C02671=1902.025400,220.027500,-703.720300,90.647653,-0.183346,-0.000000
C02672=1936.034400,220.049100,-703.720300,90.647653,-0.183346,-0.000000
C02673=1947.501800,220.061300,-703.720300,90.647653,-0.183346,-0.000000
C02674=1883.123400,220.069100,-703.720300,90.647653,-0.183346,-0.000000
C02675=2183.365000,220.088300,-703.720300,90.647653,-0.183346,-0.000000
C02676=1917.413700,220.121800,-703.720300,90.647653,-0.183346,-0.000000
C02677=1873.196800,220.137600,-703.720300,90.647653,-0.183346,-0.000000
C02678=2183.234000,220.175800,-703.720300,90.647653,-0.183346,-0.000000
C02679=1859.481200,220.212300,-703.720300,90.647653,-0.183346,-0.000000
C02680=1876.167800,220.252900,-703.720300,90.647653,-0.183346,-0.000000
C02681=2184.784300,220.282900,-703.720300,90.647653,-0.183346,-0.000000
C02682=1857.137100,220.330000,-703.720300,90.647653,-0.183346,-0.000000
C02683=1851.834100,220.481200,-703.720300,90.647653,-0.183346,-0.000000
C02684=1843.863200,220.525500,-703.720300,90.647653,-0.183346,-0.000000
C02685=1838.599500,220.632600,-703.720300,90.647653,-0.183346,-0.000000
C02686=1828.269700,220.740000,-703.720300,90.647653,-0.183346,-0.000000
C02687=1824.941700,220.777500,-703.720300,90.647653,-0.183346,-0.000000
C02688=1794.350900,220.933900,-703.720300,90.647653,-0.183346,-0.000000
C02689=1816.456800,221.034500,-703.720300,90.647653,-0.183346,-0.000000
C02690=1818.517400,221.113300,-703.720300,90.647653,-0.183346,-0.000000
C02691=1794.707900,221.180900,-703.720300,90.647653,-0.183346,-0.000000
C02692=1804.703800,221.313700,-703.720300,90.647653,-0.183346,-0.000000
C02693=1808.802700,221.407900,-703.720300,90.647653,-0.183346,-0.000000
C02694=1797.626000,221.486500,-703.720300,90.647653,-0.183346,-0.000000
C02695=1799.014100,221.558000,-703.720300,90.647653,-0.183346,-0.000000
C02696=1799.493300,221.627400,-753.720300,90.647653,-0.183346,-0.000000
C02697=1803.199100,221.533000,-753.720300,90.647653,-0.183346,-0.000000
C02698=1804.482800,221.440400,-753.720300,90.647653,-0.183346,-0.000000
C02699=1806.656400,221.406800,-753.720300,90.647653,-0.183346,-0.000000
C02700=1812.999200,221.332300,-753.720300,90.647653,-0.183346,-0.000000
C02701=1810.456500,221.261700,-753.720300,90.647653,-0.183346,-0.000000
C02702=1819.601700,221.167700,-753.720300,90.647653,-0.183346,-0.000000
C02703=1828.737100,221.094100,-753.720300,90.647653,-0.183346,-0.000000
C02704=1826.975900,220.979200,-753.720300,90.647653,-0.183346,-0.000000
C02705=1827.057400,220.918400,-753.720300,90.647653,-0.183346,-0.000000
C02706=1840.828400,220.793700,-753.720300,90.647653,-0.183346,-0.000000
C02707=1843.616100,220.652500,-753.720300,90.647653,-0.183346,-0.000000
C02708=1848.358800,220.494700,-753.720300,90.647653,-0.183346,-0.000000
C02709=1855.244300,220.394700,-753.720300,90.647653,-0.183346,-0.000000
C02710=1859.292000,220.310300,-753.720300,90.647653,-0.183346,-0.000000
C02711=1861.936400,220.207200,-753.720300,90.647653,-0.183346,-0.000000
C02712=1863.356300,220.145800,-753.720300,90.647653,-0.183346,-0.000000
C02713=1880.995500,220.085300,-753.720300,90.647653,-0.183346,-0.000000
C02714=1886.645600,220.008400,-753.720300,90.647653,-0.183346,-0.000000
C02715=1888.756600,219.930200,-753.720300,90.647653,-0.183346,-0.000000
C02716=1888.087000,219.894400,-753.720300,90.647653,-0.183346,-0.000000
C02717=1901.700500,219.846400,-753.720300,90.647653,-0.183346,-0.000000
C02718=1899.152700,219.782200,-753.720300,90.647653,-0.183346,-0.000000
C02719=1896.702700,219.751800,-753.720300,90.647653,-0.183346,-0.000000
C02720=2159.599800,219.718700,-753.720300,90.647653,-0.183346,-0.000000
C02721=1898.573400,219.689000,-753.720300,90.647653,-0.183346,-0.000000
C02722=2190.999200,219.661600,-753.720300,90.647653,-0.183346,-0.000000
C02723=1908.414200,219.628500,-753.720300,90.647653,-0.183346,-0.000000
C02724=2178.349900,219.615200,-753.720300,90.647653,-0.183346,-0.000000
C02725=1918.020800,219.596800,-753.720300,90.647653,-0.183346,-0.000000
C02726=2162.631500,219.573400,-753.720300,90.647653,-0.183346,-0.000000
C02727=2163.426800,219.563600,-753.720300,90.647653,-0.183346,-0.000000
C02728=1918.500400,219.534600,-753.720300,90.647653,-0.183346,-0.000000
C02729=2179.089400,219.517700,-753.720300,90.647653,-0.183346,-0.000000
C02730=2153.107500,219.504900,-753.720300,90.647653,-0.183346,-0.000000
C02731=1927.323900,219.499800,-753.720300,90.647653,-0.183346,-0.000000
C02732=1962.897900,219.487000,-753.720300,90.647653,-0.183346,-0.000000
C02733=2152.945000,219.474800,-753.720300,90.647653,-0.183346,-0.000000
C02734=1923.549800,219.465000,-753.720300,90.647653,-0.183346,-0.000000
C02735=2167.654000,219.443400,-753.720300,90.647653,-0.183346,-0.000000
C02736=2127.277400,219.427200,-753.720300,90.647653,-0.183346,-0.000000
C02737=2157.455000,219.411600,-753.720300,90.647653,-0.183346,-0.000000
C02738=2181.610100,219.398800,-753.720300,90.647653,-0.183346,-0.000000
C02739=1942.548000,219.387600,-753.720300,90.647653,-0.183346,-0.000000
C02740=1942.914300,219.375500,-753.720300,90.647653,-0.183346,-0.000000
C02741=2146.459000,219.360600,-753.720300,90.647653,-0.183346,-0.000000
C02742=1943.803100,219.342400,-753.720300,90.647653,-0.183346,-0.000000
C02743=2144.906500,219.324500,-753.720300,90.647653,-0.183346,-0.000000
C02744=1955.055200,219.314300,-753.720300,90.647653,-0.183346,-0.000000
C02745=2126.347200,219.294700,-753.720300,90.647653,-0.183346,-0.000000
C02746=1945.956100,219.289000,-753.720300,90.647653,-0.183346,-0.000000
C02747=1962.818800,219.279900,-753.720300,90.647653,-0.183346,-0.000000
C02748=1984.835000,219.262300,-753.720300,90.647653,-0.183346,-0.000000
C02749=1961.384800,219.248800,-753.720300,90.647653,-0.183346,-0.000000
C02750=2132.790400,219.237600,-753.720300,90.647653,-0.183346,-0.000000
C02751=2000.726200,219.227200,-753.720300,90.647653,-0.183346,-0.000000
C02752=1953.023500,219.217700,-753.720300,90.647653,-0.183346,-0.000000
C02753=2110.038700,219.210900,-753.720300,90.647653,-0.183346,-0.000000
C02754=2009.596400,219.203500,-753.720300,90.647653,-0.183346,-0.000000
C02755=2132.660700,219.194400,-753.720300,90.647653,-0.183346,-0.000000
C02756=2014.251400,219.182900,-753.720300,90.647653,-0.183346,-0.000000
C02757=2125.162500,219.168400,-753.720300,90.647653,-0.183346,-0.000000
C02758=2104.208600,219.149400,-753.720300,90.647653,-0.183346,-0.000000
C02759=2129.301800,219.144000,-753.720300,90.647653,-0.183346,-0.000000
C02760=2071.342900,219.139600,-753.720300,90.647653,-0.183346,-0.000000
C02761=2057.003000,219.115300,-753.720300,90.647653,-0.183346,-0.000000
C02762=2060.754400,219.103200,-753.720300,90.647653,-0.183346,-0.000000
C02763=1975.391800,219.089300,-753.720300,90.647653,-0.183346,-0.000000
C02764=2041.350200,219.082200,-753.720300,90.647653,-0.183346,-0.000000
C02765=2058.370700,219.077800,-753.720300,90.647653,-0.183346,-0.000000
C02766=2014.830600,219.072400,-753.720300,90.647653,-0.183346,-0.000000
C02767=1968.445400,219.059600,-753.720300,90.647653,-0.183346,-0.000000
C02768=2054.250900,219.044000,-753.720300,90.647653,-0.183346,-0.000000
C02769=2104.495100,219.038300,-753.720300,90.647653,-0.183346,-0.000000
C02770=2082.338100,219.029200,-753.720300,90.647653,-0.183346,-0.000000
C02771=2027.175600,219.021400,-753.720300,90.647653,-0.183346,-0.000000
C02772=1997.599100,219.010600,-753.720300,90.647653,-0.183346,-0.000000
C02773=2074.350800,218.995400,-753.720300,90.647653,-0.183346,-0.000000
C02774=2088.675300,218.990300,-753.720300,90.647653,-0.183346,-0.000000
C02775=2052.849400,218.981200,-753.720300,90.647653,-0.183346,-0.000000
C02776=2096.650800,218.977100,-753.720300,90.647653,-0.183346,-0.000000
C02777=2021.793300,218.962300,-753.720300,90.647653,-0.183346,-0.000000
C02778=2024.376200,218.935600,-753.720300,90.647653,-0.183346,-0.000000
C02779=2084.858800,218.917700,-753.720300,90.647653,-0.183346,-0.000000
C02780=2037.732300,218.909600,-753.720300,90.647653,-0.183346,-0.000000
C02781=2066.030000,218.889600,-753.720300,90.647653,-0.183346,-0.000000
C02782=2093.060000,218.868000,-753.720300,90.647653,-0.183346,-0.000000
C02783=2057.961700,218.804300,-753.720300,90.647653,-0.183346,-0.000000
C02784=2072.588600,218.737900,-803.720300,90.647653,-0.183346,-0.000000
C02785=2061.790300,218.784200,-803.720300,90.647653,-0.183346,-0.000000
C02786=2060.744300,218.794000,-803.720300,90.647653,-0.183346,-0.000000
C02787=1998.766800,218.818700,-803.720300,90.647653,-0.183346,-0.000000
C02788=2060.686400,218.861300,-803.720300,90.647653,-0.183346,-0.000000
C02789=2096.522100,218.870400,-803.720300,90.647653,-0.183346,-0.000000
C02790=2032.427400,218.885600,-803.720300,90.647653,-0.183346,-0.000000
C02791=2103.743000,218.891700,-803.720300,90.647653,-0.183346,-0.000000
C02792=2019.306500,218.901100,-803.720300,90.647653,-0.183346,-0.000000
C02793=2031.745000,218.913300,-803.720300,90.647653,-0.183346,-0.000000
C02794=2088.498600,218.920400,-803.720300,90.647653,-0.183346,-0.000000
C02795=2037.798100,218.927100,-803.720300,90.647653,-0.183346,-0.000000
C02796=2014.134600,218.935900,-803.720300,90.647653,-0.183346,-0.000000
C02797=2099.616700,218.942000,-803.720300,90.647653,-0.183346,-0.000000
C02798=2045.679500,218.947800,-803.720300,90.647653,-0.183346,-0.000000
C02799=2076.855800,218.951800,-803.720300,90.647653,-0.183346,-0.000000
C02800=2071.493100,218.956200,-803.720300,90.647653,-0.183346,-0.000000
C02801=1988.395700,218.967300,-803.720300,90.647653,-0.183346,-0.000000
C02802=2111.290700,218.977500,-803.720300,90.647653,-0.183346,-0.000000
C02803=2118.179700,218.990000,-803.720300,90.647653,-0.183346,-0.000000
C02804=2105.312500,218.993700,-803.720300,90.647653,-0.183346,-0.000000
C02805=2049.201500,218.998800,-803.720300,90.647653,-0.183346,-0.000000
C02806=2122.327100,219.005500,-803.720300,90.647653,-0.183346,-0.000000
C02807=1998.043700,219.019700,-803.720300,90.647653,-0.183346,-0.000000
C02808=2158.716300,219.030900,-803.720300,90.647653,-0.183346,-0.000000
C02809=2101.906500,219.037600,-803.720300,90.647653,-0.183346,-0.000000
C02810=2041.862200,219.043400,-803.720300,90.647653,-0.183346,-0.000000
C02811=2113.073500,219.050500,-803.720300,90.647653,-0.183346,-0.000000
C02812=2130.536300,219.062600,-803.720300,90.647653,-0.183346,-0.000000
C02813=1989.990900,219.069400,-803.720300,90.647653,-0.183346,-0.000000
C02814=2153.711100,219.082200,-803.720300,90.647653,-0.183346,-0.000000
C02815=2103.281100,219.093000,-803.720300,90.647653,-0.183346,-0.000000
C02816=1978.401700,219.105400,-803.720300,90.647653,-0.183346,-0.000000
C02817=2108.215500,219.112300,-803.720300,90.647653,-0.183346,-0.000000
C02818=2116.807500,219.121100,-803.720300,90.647653,-0.183346,-0.000000
C02819=2167.389500,219.129500,-803.720300,90.647653,-0.183346,-0.000000
C02820=1968.224900,219.147100,-803.720300,90.647653,-0.183346,-0.000000
C02821=1980.356400,219.152100,-803.720300,90.647653,-0.183346,-0.000000
C02822=2012.286700,219.161300,-803.720300,90.647653,-0.183346,-0.000000
C02823=1979.045200,219.176100,-803.720300,90.647653,-0.183346,-0.000000
C02824=2132.626900,219.183900,-803.720300,90.647653,-0.183346,-0.000000
C02825=2138.833300,219.206700,-803.720300,90.647653,-0.183346,-0.000000
C02826=2189.419500,219.215000,-803.720300,90.647653,-0.183346,-0.000000
C02827=2163.932900,219.221100,-803.720300,90.647653,-0.183346,-0.000000
C02828=1973.290700,219.229500,-803.720300,90.647653,-0.183346,-0.000000
C02829=1962.589400,219.234900,-803.720300,90.647653,-0.183346,-0.000000
C02830=2140.348900,219.251500,-803.720300,90.647653,-0.183346,-0.000000
C02831=1966.086800,219.259900,-803.720300,90.647653,-0.183346,-0.000000
C02832=2146.072100,219.278200,-803.720300,90.647653,-0.183346,-0.000000
C02833=1944.019200,219.307900,-803.720300,90.647653,-0.183346,-0.000000
C02834=2164.122900,219.335600,-803.720300,90.647653,-0.183346,-0.000000
C02835=2179.267500,219.347800,-803.720300,90.647653,-0.183346,-0.000000
C02836=1958.782200,219.356200,-803.720300,90.647653,-0.183346,-0.000000
C02837=1950.731800,219.377800,-803.720300,90.647653,-0.183346,-0.000000
C02838=1939.923400,219.405900,-803.720300,90.647653,-0.183346,-0.000000
C02839=1952.384300,219.433200,-803.720300,90.647653,-0.183346,-0.000000
C02840=1939.916500,219.453500,-803.720300,90.647653,-0.183346,-0.000000
C02841=1924.529600,219.509300,-803.720300,90.647653,-0.183346,-0.000000
C02842=1931.308400,219.530200,-803.720300,90.647653,-0.183346,-0.000000
C02843=1915.280200,219.568700,-803.720300,90.647653,-0.183346,-0.000000
C02844=1925.417000,219.624800,-803.720300,90.647653,-0.183346,-0.000000
C02845=1938.538700,219.697400,-803.720300,90.647653,-0.183346,-0.000000
C02846=1916.231700,219.759600,-803.720300,90.647653,-0.183346,-0.000000
C02847=1905.662800,219.803200,-803.720300,90.647653,-0.183346,-0.000000
C02848=1907.860700,219.882600,-803.720300,90.647653,-0.183346,-0.000000
C02849=1891.452900,219.963300,-803.720300,90.647653,-0.183346,-0.000000
C02850=1897.806200,220.044700,-803.720300,90.647653,-0.183346,-0.000000
C02851=1877.774400,220.141500,-803.720300,90.647653,-0.183346,-0.000000
C02852=1889.906800,220.208900,-803.720300,90.647653,-0.183346,-0.000000
C02853=1873.599400,220.241000,-803.720300,90.647653,-0.183346,-0.000000
C02854=1871.595600,220.341000,-803.720300,90.647653,-0.183346,-0.000000
C02855=1877.964600,220.428500,-803.720300,90.647653,-0.183346,-0.000000
C02856=1863.088700,220.547800,-803.720300,90.647653,-0.183346,-0.000000
C02857=1857.730100,220.604900,-803.720300,90.647653,-0.183346,-0.000000
C02858=1845.662400,220.779600,-803.720300,90.647653,-0.183346,-0.000000
C02859=1845.976100,220.851500,-803.720300,90.647653,-0.183346,-0.000000
C02860=1839.138000,220.982300,-803.720300,90.647653,-0.183346,-0.000000
C02861=1829.338300,221.025500,-803.720300,90.647653,-0.183346,-0.000000
C02862=1794.450600,221.067700,-803.720300,90.647653,-0.183346,-0.000000
C02863=1837.453500,221.120100,-803.720300,90.647653,-0.183346,-0.000000
C02864=1823.782100,221.184000,-803.720300,90.647653,-0.183346,-0.000000
C02865=1816.928300,221.265000,-803.720300,90.647653,-0.183346,-0.000000
C02866=1816.898000,221.328600,-803.720300,90.647653,-0.183346,-0.000000
C02867=1807.872100,221.425900,-803.720300,90.647653,-0.183346,-0.000000
C02868=1812.030900,221.466400,-803.720300,90.647653,-0.183346,-0.000000
C02869=1797.540300,221.537700,-803.720300,90.647653,-0.183346,-0.000000
C02870=1797.919500,221.574000,-803.720300,90.647653,-0.183346,-0.000000
C02871=1798.307500,221.652200,-803.720300,90.647653,-0.183346,-0.000000
C02872=1798.204800,221.824500,-853.720300,90.647653,-0.183346,-0.000000
C02873=1801.321900,221.694400,-853.720300,90.647653,-0.183346,-0.000000
C02874=1803.359500,221.606900,-853.720300,90.647653,-0.183346,-0.000000
C02875=1796.778200,221.518400,-853.720300,90.647653,-0.183346,-0.000000
C02876=1810.824300,221.446100,-853.720300,90.647653,-0.183346,-0.000000
C02877=1812.569900,221.372100,-853.720300,90.647653,-0.183346,-0.000000
C02878=1813.958700,221.320100,-853.720300,90.647653,-0.183346,-0.000000
C02879=1816.060500,221.201900,-853.720300,90.647653,-0.183346,-0.000000
C02880=1822.471300,221.136300,-853.720300,90.647653,-0.183346,-0.000000
C02881=1816.917900,221.114700,-853.720300,90.647653,-0.183346,-0.000000
C02882=1843.384000,220.988000,-853.720300,90.647653,-0.183346,-0.000000
C02883=1841.543700,220.882300,-853.720300,90.647653,-0.183346,-0.000000
C02884=1842.988700,220.787700,-853.720300,90.647653,-0.183346,-0.000000
C02885=1849.877000,220.765400,-853.720300,90.647653,-0.183346,-0.000000
C02886=1858.351200,220.668100,-853.720300,90.647653,-0.183346,-0.000000
C02887=1864.384500,220.598800,-853.720300,90.647653,-0.183346,-0.000000
C02888=1864.226300,220.572800,-853.720300,90.647653,-0.183346,-0.000000
C02889=1884.340500,220.452200,-853.720300,90.647653,-0.183346,-0.000000
C02890=1866.225600,220.418700,-853.720300,90.647653,-0.183346,-0.000000
C02891=1874.781700,220.325800,-853.720300,90.647653,-0.183346,-0.000000
C02892=1888.846900,220.302500,-853.720300,90.647653,-0.183346,-0.000000
C02893=1890.867400,220.245800,-853.720300,90.647653,-0.183346,-0.000000
C02894=1896.806300,220.168700,-853.720300,90.647653,-0.183346,-0.000000
C02895=1904.238600,220.121800,-853.720300,90.647653,-0.183346,-0.000000
C02896=1933.711600,220.093100,-853.720300,90.647653,-0.183346,-0.000000
C02897=1904.412600,220.009600,-853.720300,90.647653,-0.183346,-0.000000
C02898=1912.942200,219.983900,-853.720300,90.647653,-0.183346,-0.000000
C02899=1923.653300,219.915300,-853.720300,90.647653,-0.183346,-0.000000
C02900=1952.154200,219.830900,-853.720300,90.647653,-0.183346,-0.000000
C02901=1953.177900,219.787300,-853.720300,90.647653,-0.183346,-0.000000
C02902=1946.822900,219.765300,-853.720300,90.647653,-0.183346,-0.000000
C02903=1929.570200,219.735600,-853.720300,90.647653,-0.183346,-0.000000
C02904=1937.309500,219.673800,-853.720300,90.647653,-0.183346,-0.000000
C02905=1937.928700,219.640000,-853.720300,90.647653,-0.183346,-0.000000
C02906=2046.786800,219.592700,-853.720300,90.647653,-0.183346,-0.000000
C02907=1962.466300,219.525800,-853.720300,90.647653,-0.183346,-0.000000
C02908=1984.675200,219.491300,-853.720300,90.647653,-0.183346,-0.000000
C02909=1980.669800,219.452500,-853.720300,90.647653,-0.183346,-0.000000
C02910=1957.287600,219.413300,-853.720300,90.647653,-0.183346,-0.000000
C02911=1990.034400,219.407900,-853.720300,90.647653,-0.183346,-0.000000
C02912=2000.277100,219.357200,-853.720300,90.647653,-0.183346,-0.000000
C02913=1982.379600,219.320700,-853.720300,90.647653,-0.183346,-0.000000
C02914=2009.503800,219.300100,-853.720300,90.647653,-0.183346,-0.000000
C02915=2024.065300,219.287600,-853.720300,90.647653,-0.183346,-0.000000
C02916=2121.036700,219.277500,-853.720300,90.647653,-0.183346,-0.000000
C02917=2054.858100,219.232900,-853.720300,90.647653,-0.183346,-0.000000
C02918=2038.027500,219.216700,-853.720300,90.647653,-0.183346,-0.000000
C02919=2082.814900,219.200600,-853.720300,90.647653,-0.183346,-0.000000
C02920=1988.741400,219.188600,-853.720300,90.647653,-0.183346,-0.000000
C02921=2066.833000,219.181900,-853.720300,90.647653,-0.183346,-0.000000
C02922=2187.536400,219.174400,-853.720300,90.647653,-0.183346,-0.000000
C02923=2005.816200,219.153200,-853.720300,90.647653,-0.183346,-0.000000
C02924=2086.585100,219.138300,-853.720300,90.647653,-0.183346,-0.000000
C02925=2181.706300,219.132600,-853.720300,90.647653,-0.183346,-0.000000
C02926=2164.749100,219.125800,-853.720300,90.647653,-0.183346,-0.000000
C02927=2178.936800,219.119700,-853.720300,90.647653,-0.183346,-0.000000
C02928=2178.300300,219.107900,-853.720300,90.647653,-0.183346,-0.000000
C02929=1994.649700,219.099800,-853.720300,90.647653,-0.183346,-0.000000
C02930=1997.640300,219.092000,-853.720300,90.647653,-0.183346,-0.000000
C02931=2027.654600,219.084600,-853.720300,90.647653,-0.183346,-0.000000
C02932=2071.270700,219.078500,-853.720300,90.647653,-0.183346,-0.000000
C02933=2107.465400,219.071700,-853.720300,90.647653,-0.183346,-0.000000
C02934=2171.342000,219.061900,-853.720300,90.647653,-0.183346,-0.000000
C02935=2005.844500,219.057200,-853.720300,90.647653,-0.183346,-0.000000
C02936=2061.146900,219.048800,-853.720300,90.647653,-0.183346,-0.000000
C02937=2091.887500,219.042300,-853.720300,90.647653,-0.183346,-0.000000
C02938=2126.755700,219.031500,-853.720300,90.647653,-0.183346,-0.000000
C02939=2141.745600,219.024800,-853.720300,90.647653,-0.183346,-0.000000
C02940=2049.929600,219.015000,-853.720300,90.647653,-0.183346,-0.000000
C02941=2016.646200,219.011300,-853.720300,90.647653,-0.183346,-0.000000
C02942=2096.581400,219.008200,-853.720300,90.647653,-0.183346,-0.000000
C02943=2146.224700,218.999400,-853.720300,90.647653,-0.183346,-0.000000
C02944=2169.186900,218.994000,-853.720300,90.647653,-0.183346,-0.000000
C02945=2155.428400,218.980500,-853.720300,90.647653,-0.183346,-0.000000
C02946=2135.209300,218.964000,-853.720300,90.647653,-0.183346,-0.000000
C02947=2045.472400,218.951500,-853.720300,90.647653,-0.183346,-0.000000
C02948=2090.833200,218.942300,-853.720300,90.647653,-0.183346,-0.000000
C02949=2072.000200,218.937300,-853.720300,90.647653,-0.183346,-0.000000
C02950=2108.548700,218.918400,-853.720300,90.647653,-0.183346,-0.000000
C02951=2058.766300,218.909200,-853.720300,90.647653,-0.183346,-0.000000
C02952=2188.558300,218.899800,-853.720300,90.647653,-0.183346,-0.000000
C02953=2113.179100,218.886600,-853.720300,90.647653,-0.183346,-0.000000
C02954=2114.456500,218.868000,-853.720300,90.647653,-0.183346,-0.000000
C02955=2141.480300,218.844700,-853.720300,90.647653,-0.183346,-0.000000
C02956=2157.691900,218.778500,-853.720300,90.647653,-0.183346,-0.000000
C02957=2182.358100,218.678800,-853.720300,90.647653,-0.183346,-0.000000
C02958=2191.986300,218.384600,-853.720300,90.647653,-0.183346,-0.000000
C02959=1844.503600,-183.911800,-453.729100,88.350092,-0.177617,0.005730
C02960=2102.179900,-183.692800,-453.729100,88.350092,-0.177617,0.005730
C02961=2105.483700,-183.499400,-453.729100,88.350092,-0.177617,0.005730
C02962=1867.597200,-183.372200,-453.729100,88.350092,-0.177617,0.005730
C02963=2040.843900,-183.333400,-453.729100,88.350092,-0.177617,0.005730
C02964=2098.536500,-183.311400,-453.729100,88.350092,-0.177617,0.005730
C02965=2076.129600,-183.225300,-453.729100,88.350092,-0.177617,0.005730
C02966=2054.784300,-183.195200,-453.729100,88.350092,-0.177617,0.005730
C02967=1928.436500,-183.147900,-453.729100,88.350092,-0.177617,0.005730
C02968=1952.498400,-183.085100,-453.729100,88.350092,-0.177617,0.005730
C02969=2042.123700,-183.045500,-453.729100,88.350092,-0.177617,0.005730
C02970=1972.749900,-182.957700,-453.729100,88.350092,-0.177617,0.005730
C02971=1920.402200,-182.151600,-503.729100,88.350092,-0.177617,0.005730
C02972=1910.020800,-182.237700,-503.729100,88.350092,-0.177617,0.005730
C02973=1865.559600,-182.301600,-503.729100,88.350092,-0.177617,0.005730
C02974=1869.102600,-182.378600,-503.729100,88.350092,-0.177617,0.005730
C02975=1915.063200,-182.406300,-503.729100,88.350092,-0.177617,0.005730
C02976=1860.422400,-182.470200,-503.729100,88.350092,-0.177617,0.005730
C02977=1936.524200,-182.488400,-503.729100,88.350092,-0.177617,0.005730
C02978=1997.214500,-182.508000,-503.729100,88.350092,-0.177617,0.005730
C02979=2018.653800,-182.520500,-503.729100,88.350092,-0.177617,0.005730
C02980=1932.008800,-182.551900,-503.729100,88.350092,-0.177617,0.005730
C02981=2023.031800,-182.571200,-503.729100,88.350092,-0.177617,0.005730
C02982=2015.175200,-182.574200,-503.729100,88.350092,-0.177617,0.005730
C02983=1956.558200,-182.592800,-503.729100,88.350092,-0.177617,0.005730
C02984=2088.791200,-182.625900,-503.729100,88.350092,-0.177617,0.005730
C02985=1856.430200,-182.636100,-503.729100,88.350092,-0.177617,0.005730
C02986=1868.122100,-182.664400,-503.729100,88.350092,-0.177617,0.005730
C02987=1954.832200,-182.687400,-503.729100,88.350092,-0.177617,0.005730
C02988=1979.253000,-182.706300,-503.729100,88.350092,-0.177617,0.005730
C02989=2079.993900,-182.726600,-503.729100,88.350092,-0.177617,0.005730
C02990=1848.373900,-182.742100,-503.729100,88.350092,-0.177617,0.005730
C02991=1897.192200,-182.754300,-503.729100,88.350092,-0.177617,0.005730
C02992=2075.658700,-182.763400,-503.729100,88.350092,-0.177617,0.005730
C02993=2078.649700,-182.781000,-503.729100,88.350092,-0.177617,0.005730
C02994=1866.835000,-182.792500,-503.729100,88.350092,-0.177617,0.005730
C02995=1896.216300,-182.810700,-503.729100,88.350092,-0.177617,0.005730
C02996=2005.012300,-182.828300,-503.729100,88.350092,-0.177617,0.005730
C02997=2095.740700,-182.834400,-503.729100,88.350092,-0.177617,0.005730
C02998=2002.510100,-182.848200,-503.729100,88.350092,-0.177617,0.005730
C02999=1972.794600,-182.868200,-503.729100,88.350092,-0.177617,0.005730
C03000=2123.363400,-182.881000,-503.729100,88.350092,-0.177617,0.005730
C03001=2093.091200,-182.896900,-503.729100,88.350092,-0.177617,0.005730
C03002=2130.634100,-182.905700,-503.729100,88.350092,-0.177617,0.005730
C03003=1883.316300,-182.917100,-503.729100,88.350092,-0.177617,0.005730
C03004=1947.839000,-182.931300,-503.729100,88.350092,-0.177617,0.005730
C03005=1984.973400,-182.935700,-503.729100,88.350092,-0.177617,0.005730
C03006=2087.406800,-182.947500,-503.729100,88.350092,-0.177617,0.005730
C03007=1906.237700,-182.958400,-503.729100,88.350092,-0.177617,0.005730
C03008=2054.050600,-182.967500,-503.729100,88.350092,-0.177617,0.005730
C03009=2024.974500,-182.976300,-503.729100,88.350092,-0.177617,0.005730
C03010=2115.214800,-182.984000,-503.729100,88.350092,-0.177617,0.005730
C03011=1931.895900,-182.996200,-503.729100,88.350092,-0.177617,0.005730
C03012=2090.852000,-183.001800,-503.729100,88.350092,-0.177617,0.005730
C03013=1944.513600,-183.014100,-503.729100,88.350092,-0.177617,0.005730
C03014=2020.788800,-183.021800,-503.729100,88.350092,-0.177617,0.005730
C03015=2192.002800,-183.030300,-503.729100,88.350092,-0.177617,0.005730
C03016=1992.711900,-183.041500,-503.729100,88.350092,-0.177617,0.005730
C03017=2116.416200,-183.046200,-503.729100,88.350092,-0.177617,0.005730
C03018=2149.219900,-183.051900,-503.729100,88.350092,-0.177617,0.005730
C03019=2025.231500,-183.056700,-503.729100,88.350092,-0.177617,0.005730
C03020=2179.699900,-183.062800,-503.729100,88.350092,-0.177617,0.005730
C03021=1952.937900,-183.069800,-503.729100,88.350092,-0.177617,0.005730
C03022=2025.823200,-183.073200,-503.729100,88.350092,-0.177617,0.005730
C03023=1900.850200,-183.080500,-503.729100,88.350092,-0.177617,0.005730
C03024=2082.318000,-183.090500,-503.729100,88.350092,-0.177617,0.005730
C03025=1967.121500,-183.098600,-503.729100,88.350092,-0.177617,0.005730
C03026=2141.273800,-183.105300,-503.729100,88.350092,-0.177617,0.005730
C03027=2012.174100,-183.113100,-503.729100,88.350092,-0.177617,0.005730
C03028=2069.713900,-183.122600,-503.729100,88.350092,-0.177617,0.005730
C03029=2075.940000,-183.135700,-503.729100,88.350092,-0.177617,0.005730
C03030=1912.803600,-183.141500,-503.729100,88.350092,-0.177617,0.005730
C03031=2161.003900,-183.146500,-503.729100,88.350092,-0.177617,0.005730
C03032=1987.916900,-183.148900,-503.729100,88.350092,-0.177617,0.005730
C03033=1907.835400,-183.154000,-503.729100,88.350092,-0.177617,0.005730
C03034=2184.356300,-183.163200,-503.729100,88.350092,-0.177617,0.005730
C03035=1909.521000,-183.167100,-503.729100,88.350092,-0.177617,0.005730
C03036=2169.104400,-183.173200,-503.729100,88.350092,-0.177617,0.005730
C03037=2167.713000,-183.178300,-503.729100,88.350092,-0.177617,0.005730
C03038=1864.364100,-183.181700,-503.729100,88.350092,-0.177617,0.005730
C03039=1815.055400,-183.183400,-503.729100,88.350092,-0.177617,0.005730
C03040=2022.864700,-183.191800,-503.729100,88.350092,-0.177617,0.005730
C03041=2122.878600,-183.197900,-503.729100,88.350092,-0.177617,0.005730
C03042=2078.860200,-183.204500,-503.729100,88.350092,-0.177617,0.005730
C03043=2041.006800,-183.213900,-503.729100,88.350092,-0.177617,0.005730
C03044=1803.617900,-183.216800,-503.729100,88.350092,-0.177617,0.005730
C03045=2170.640800,-183.223200,-503.729100,88.350092,-0.177617,0.005730
C03046=2033.959000,-183.226900,-503.729100,88.350092,-0.177617,0.005730
C03047=2173.908400,-183.230700,-503.729100,88.350092,-0.177617,0.005730
C03048=2188.998400,-183.237100,-503.729100,88.350092,-0.177617,0.005730
C03049=2164.107300,-183.249200,-503.729100,88.350092,-0.177617,0.005730
C03050=2186.876800,-183.255000,-503.729100,88.350092,-0.177617,0.005730
C03051=1809.229400,-183.262600,-503.729100,88.350092,-0.177617,0.005730
C03052=2094.103900,-183.266500,-503.729100,88.350092,-0.177617,0.005730
C03053=2112.401000,-183.271500,-503.729100,88.350092,-0.177617,0.005730
C03054=2046.259600,-183.281700,-503.729100,88.350092,-0.177617,0.005730
C03055=2036.649100,-183.290500,-503.729100,88.350092,-0.177617,0.005730
C03056=2021.180400,-183.295200,-503.729100,88.350092,-0.177617,0.005730
C03057=2139.838800,-183.305700,-503.729100,88.350092,-0.177617,0.005730
C03058=1878.389900,-183.315100,-503.729100,88.350092,-0.177617,0.005730
C03059=2075.564900,-183.337100,-503.729100,88.350092,-0.177617,0.005730
C03060=1820.257100,-183.355300,-503.729100,88.350092,-0.177617,0.005730
C03061=2100.825100,-183.365800,-503.729100,88.350092,-0.177617,0.005730
C03062=1838.000100,-183.374600,-503.729100,88.350092,-0.177617,0.005730
C03063=1919.496400,-183.382700,-503.729100,88.350092,-0.177617,0.005730
C03064=1847.459000,-183.397600,-503.729100,88.350092,-0.177617,0.005730
C03065=1810.340900,-183.421700,-503.729100,88.350092,-0.177617,0.005730
C03066=1804.173400,-183.438800,-503.729100,88.350092,-0.177617,0.005730
C03067=2143.420800,-183.472600,-503.729100,88.350092,-0.177617,0.005730
C03068=1809.991000,-183.536800,-503.729100,88.350092,-0.177617,0.005730
C03069=1861.800900,-183.622200,-503.729100,88.350092,-0.177617,0.005730
C03070=1830.538800,-183.688400,-503.729100,88.350092,-0.177617,0.005730
C03071=1795.005800,-183.716800,-503.729100,88.350092,-0.177617,0.005730
C03072=1845.825000,-183.769200,-503.729100,88.350092,-0.177617,0.005730
C03073=1817.353000,-183.887800,-503.729100,88.350092,-0.177617,0.005730
C03074=1800.477100,-183.922600,-503.729100,88.350092,-0.177617,0.005730
C03075=1804.847200,-184.149600,-503.729100,88.350092,-0.177617,0.005730
C03076=2191.964500,-184.111100,-553.729100,88.350092,-0.177617,0.005730
C03077=2188.007100,-183.260700,-553.729100,88.350092,-0.177617,0.005730
C03078=2188.974300,-183.181300,-553.729100,88.350092,-0.177617,0.005730
C03079=2182.610900,-183.132700,-553.729100,88.350092,-0.177617,0.005730
C03080=2180.041800,-183.063800,-553.729100,88.350092,-0.177617,0.005730
C03081=2165.917900,-183.039300,-553.729100,88.350092,-0.177617,0.005730
C03082=2170.273100,-182.998200,-553.729100,88.350092,-0.177617,0.005730
C03083=2155.198200,-182.972500,-553.729100,88.350092,-0.177617,0.005730
C03084=2138.395800,-182.940100,-553.729100,88.350092,-0.177617,0.005730
C03085=1811.107100,-182.911400,-553.729100,88.350092,-0.177617,0.005730
C03086=2170.505900,-182.875900,-553.729100,88.350092,-0.177617,0.005730
C03087=2152.789400,-182.835400,-553.729100,88.350092,-0.177617,0.005730
C03088=2172.181700,-182.784000,-553.729100,88.350092,-0.177617,0.005730
C03089=1812.654600,-182.750900,-553.729100,88.350092,-0.177617,0.005730
C03090=1803.653100,-182.728600,-553.729100,88.350092,-0.177617,0.005730
C03091=2166.890500,-182.710400,-553.729100,88.350092,-0.177617,0.005730
C03092=1835.091500,-182.684400,-553.729100,88.350092,-0.177617,0.005730
C03093=2177.309900,-182.629600,-553.729100,88.350092,-0.177617,0.005730
C03094=2099.031800,-182.604300,-553.729100,88.350092,-0.177617,0.005730
C03095=2128.420500,-182.542100,-553.729100,88.350092,-0.177617,0.005730
C03096=1807.981300,-182.526300,-553.729100,88.350092,-0.177617,0.005730
C03097=2163.367400,-182.508000,-553.729100,88.350092,-0.177617,0.005730
C03098=1819.757300,-182.469500,-553.729100,88.350092,-0.177617,0.005730
C03099=2062.562400,-182.447900,-553.729100,88.350092,-0.177617,0.005730
C03100=1835.598300,-182.412100,-553.729100,88.350092,-0.177617,0.005730
C03101=2143.515600,-182.391500,-553.729100,88.350092,-0.177617,0.005730
C03102=1814.872400,-182.369200,-553.729100,88.350092,-0.177617,0.005730
C03103=2005.611900,-182.341100,-553.729100,88.350092,-0.177617,0.005730
C03104=1813.637200,-182.327600,-553.729100,88.350092,-0.177617,0.005730
C03105=2019.288000,-182.313700,-553.729100,88.350092,-0.177617,0.005730
C03106=1934.174000,-182.290800,-553.729100,88.350092,-0.177617,0.005730
C03107=1813.756700,-182.274200,-553.729100,88.350092,-0.177617,0.005730
C03108=2037.099100,-182.249600,-553.729100,88.350092,-0.177617,0.005730
C03109=1994.144600,-182.237700,-553.729100,88.350092,-0.177617,0.005730
C03110=1820.480500,-182.223900,-553.729100,88.350092,-0.177617,0.005730
C03111=1971.012000,-182.205300,-553.729100,88.350092,-0.177617,0.005730
C03112=1870.182400,-182.187400,-553.729100,88.350092,-0.177617,0.005730
C03113=1991.177200,-182.172000,-553.729100,88.350092,-0.177617,0.005730
C03114=2130.194200,-182.157000,-553.729100,88.350092,-0.177617,0.005730
C03115=2033.998100,-182.138700,-553.729100,88.350092,-0.177617,0.005730
C03116=2113.072300,-182.096200,-553.729100,88.350092,-0.177617,0.005730
C03117=2077.424400,-182.082700,-553.729100,88.350092,-0.177617,0.005730
C03118=2156.235800,-182.066100,-553.729100,88.350092,-0.177617,0.005730
C03119=1865.039900,-182.057000,-553.729100,88.350092,-0.177617,0.005730
C03120=1986.643200,-182.040100,-553.729100,88.350092,-0.177617,0.005730
C03121=1976.798400,-182.020500,-553.729100,88.350092,-0.177617,0.005730
C03122=1895.618700,-181.994400,-553.729100,88.350092,-0.177617,0.005730
C03123=1823.673200,-181.985000,-553.729100,88.350092,-0.177617,0.005730
C03124=2094.327100,-181.977300,-553.729100,88.350092,-0.177617,0.005730
C03125=1875.441200,-181.965400,-553.729100,88.350092,-0.177617,0.005730
C03126=2073.346400,-181.942500,-553.729100,88.350092,-0.177617,0.005730
C03127=1923.389300,-181.921500,-553.729100,88.350092,-0.177617,0.005730
C03128=2115.435400,-181.915100,-553.729100,88.350092,-0.177617,0.005730
C03129=1841.043600,-181.893800,-553.729100,88.350092,-0.177617,0.005730
C03130=2026.103900,-181.868800,-553.729100,88.350092,-0.177617,0.005730
C03131=1849.383600,-181.849900,-553.729100,88.350092,-0.177617,0.005730
C03132=1873.769600,-181.828300,-553.729100,88.350092,-0.177617,0.005730
C03133=1970.430100,-181.802900,-553.729100,88.350092,-0.177617,0.005730
C03134=1986.516800,-181.777200,-553.729100,88.350092,-0.177617,0.005730
C03135=1834.074100,-181.755600,-553.729100,88.350092,-0.177617,0.005730
C03136=1979.139800,-181.741400,-553.729100,88.350092,-0.177617,0.005730
C03137=1846.921900,-181.724900,-553.729100,88.350092,-0.177617,0.005730
C03138=1830.389600,-181.698200,-553.729100,88.350092,-0.177617,0.005730
C03139=2134.207700,-181.686700,-553.729100,88.350092,-0.177617,0.005730
C03140=1918.709300,-181.666800,-553.729100,88.350092,-0.177617,0.005730
C03141=1872.071900,-181.650200,-553.729100,88.350092,-0.177617,0.005730
C03142=2088.570900,-181.637400,-553.729100,88.350092,-0.177617,0.005730
C03143=1998.178700,-181.621000,-553.729100,88.350092,-0.177617,0.005730
C03144=2117.331100,-181.599900,-553.729100,88.350092,-0.177617,0.005730
C03145=1891.996800,-181.585700,-553.729100,88.350092,-0.177617,0.005730
C03146=1993.884700,-181.570300,-553.729100,88.350092,-0.177617,0.005730
C03147=1876.387500,-181.549900,-553.729100,88.350092,-0.177617,0.005730
C03148=1860.150600,-181.531300,-553.729100,88.350092,-0.177617,0.005730
C03149=1947.582500,-181.520500,-553.729100,88.350092,-0.177617,0.005730
C03150=2064.434100,-181.493100,-553.729100,88.350092,-0.177617,0.005730
C03151=1983.088800,-181.449800,-553.729100,88.350092,-0.177617,0.005730
C03152=1944.574200,-181.399900,-553.729100,88.350092,-0.177617,0.005730
C03153=2027.050200,-181.378600,-553.729100,88.350092,-0.177617,0.005730
C03154=1876.947700,-181.347200,-553.729100,88.350092,-0.177617,0.005730
C03155=2053.152800,-181.337400,-553.729100,88.350092,-0.177617,0.005730
C03156=2070.966200,-181.316800,-553.729100,88.350092,-0.177617,0.005730
C03157=1953.379200,-181.303900,-553.729100,88.350092,-0.177617,0.005730
C03158=2078.228900,-181.253200,-553.729100,88.350092,-0.177617,0.005730
C03159=2033.379400,-181.233000,-553.729100,88.350092,-0.177617,0.005730
C03160=1999.573500,-181.216800,-553.729100,88.350092,-0.177617,0.005730
C03161=1934.599500,-181.202600,-553.729100,88.350092,-0.177617,0.005730
C03162=2015.064800,-181.163000,-553.729100,88.350092,-0.177617,0.005730
C03163=2104.273200,-181.129600,-553.729100,88.350092,-0.177617,0.005730
C03164=1926.720000,-181.123200,-553.729100,88.350092,-0.177617,0.005730
C03165=2099.227000,-181.093100,-553.729100,88.350092,-0.177617,0.005730
C03166=1967.145500,-181.048200,-553.729100,88.350092,-0.177617,0.005730
C03167=1956.449800,-181.025200,-553.729100,88.350092,-0.177617,0.005730
C03168=1906.504300,-180.983300,-553.729100,88.350092,-0.177617,0.005730
C03169=2021.091400,-180.967400,-553.729100,88.350092,-0.177617,0.005730
C03170=2043.605700,-180.927600,-553.729100,88.350092,-0.177617,0.005730
C03171=1944.414600,-180.891100,-553.729100,88.350092,-0.177617,0.005730
C03172=2034.040300,-180.869800,-553.729100,88.350092,-0.177617,0.005730
C03173=2050.203700,-180.843100,-553.729100,88.350092,-0.177617,0.005730
C03174=2085.765100,-180.803200,-553.729100,88.350092,-0.177617,0.005730
C03175=1974.722600,-180.782400,-553.729100,88.350092,-0.177617,0.005730
C03176=1944.999400,-180.736700,-553.729100,88.350092,-0.177617,0.005730
C03177=1955.872800,-180.706400,-553.729100,88.350092,-0.177617,0.005730
C03178=2081.715700,-180.680900,-553.729100,88.350092,-0.177617,0.005730
C03179=1977.581700,-180.565700,-553.729100,88.350092,-0.177617,0.005730
C03180=1974.065700,-179.189000,-603.729100,88.350092,-0.177617,0.005730
C03181=2005.161700,-179.293100,-603.729100,88.350092,-0.177617,0.005730
C03182=2042.143200,-179.306900,-603.729100,88.350092,-0.177617,0.005730
C03183=2075.065500,-179.330200,-603.729100,88.350092,-0.177617,0.005730
C03184=2004.413700,-179.362300,-603.729100,88.350092,-0.177617,0.005730
C03185=1967.192000,-179.379600,-603.729100,88.350092,-0.177617,0.005730
C03186=1949.349600,-179.394100,-603.729100,88.350092,-0.177617,0.005730
C03187=1934.818800,-179.419100,-603.729100,88.350092,-0.177617,0.005730
C03188=1944.173500,-179.457800,-603.729100,88.350092,-0.177617,0.005730
C03189=2074.007300,-179.488000,-603.729100,88.350092,-0.177617,0.005730
C03190=1949.106000,-179.505600,-603.729100,88.350092,-0.177617,0.005730
C03191=1924.875100,-179.526200,-603.729100,88.350092,-0.177617,0.005730
C03192=1981.213100,-179.532600,-603.729100,88.350092,-0.177617,0.005730
C03193=1976.942500,-179.568100,-603.729100,88.350092,-0.177617,0.005730
C03194=2017.620100,-179.593400,-603.729100,88.350092,-0.177617,0.005730
C03195=1946.261900,-179.620400,-603.729100,88.350092,-0.177617,0.005730
C03196=2009.088000,-179.640400,-603.729100,88.350092,-0.177617,0.005730
C03197=1972.767800,-179.647500,-603.729100,88.350092,-0.177617,0.005730
C03198=2045.617200,-179.669100,-603.729100,88.350092,-0.177617,0.005730
C03199=2109.415300,-179.712700,-603.729100,88.350092,-0.177617,0.005730
C03200=1895.828000,-179.745100,-603.729100,88.350092,-0.177617,0.005730
C03201=1933.482800,-179.778900,-603.729100,88.350092,-0.177617,0.005730
C03202=2061.268600,-179.807900,-603.729100,88.350092,-0.177617,0.005730
C03203=1990.481500,-179.821500,-603.729100,88.350092,-0.177617,0.005730
C03204=2070.421800,-179.848100,-603.729100,88.350092,-0.177617,0.005730
C03205=2075.935800,-179.866400,-603.729100,88.350092,-0.177617,0.005730
C03206=1883.908100,-179.870400,-603.729100,88.350092,-0.177617,0.005730
C03207=1981.142800,-179.880600,-603.729100,88.350092,-0.177617,0.005730
C03208=1898.735900,-179.897100,-603.729100,88.350092,-0.177617,0.005730
C03209=1965.266600,-179.921800,-603.729100,88.350092,-0.177617,0.005730
C03210=2105.758400,-179.928900,-603.729100,88.350092,-0.177617,0.005730
C03211=2058.024000,-179.952900,-603.729100,88.350092,-0.177617,0.005730
C03212=1908.589300,-179.974200,-603.729100,88.350092,-0.177617,0.005730
C03213=2117.458400,-180.018100,-603.729100,88.350092,-0.177617,0.005730
C03214=1881.728300,-180.041400,-603.729100,88.350092,-0.177617,0.005730
C03215=2031.290600,-180.065700,-603.729100,88.350092,-0.177617,0.005730
C03216=2037.875700,-180.079600,-603.729100,88.350092,-0.177617,0.005730
C03217=1905.514100,-180.122100,-603.729100,88.350092,-0.177617,0.005730
C03218=2121.415700,-180.132300,-603.729100,88.350092,-0.177617,0.005730
C03219=1936.058900,-180.152200,-603.729100,88.350092,-0.177617,0.005730
C03220=2074.834700,-180.177200,-603.729100,88.350092,-0.177617,0.005730
C03221=2005.383200,-180.203900,-603.729100,88.350092,-0.177617,0.005730
C03222=1891.110800,-180.212300,-603.729100,88.350092,-0.177617,0.005730
C03223=2013.303100,-180.251900,-603.729100,88.350092,-0.177617,0.005730
C03224=2072.969000,-180.304200,-603.729100,88.350092,-0.177617,0.005730
C03225=1919.806600,-180.313400,-603.729100,88.350092,-0.177617,0.005730
C03226=2055.183000,-180.344800,-603.729100,88.350092,-0.177617,0.005730
C03227=1975.490600,-180.355600,-603.729100,88.350092,-0.177617,0.005730
C03228=1887.334000,-180.371500,-603.729100,88.350092,-0.177617,0.005730
C03229=1873.863700,-180.388700,-603.729100,88.350092,-0.177617,0.005730
C03230=1905.720100,-180.408000,-603.729100,88.350092,-0.177617,0.005730
C03231=1885.639300,-180.438000,-603.729100,88.350092,-0.177617,0.005730
C03232=1934.848400,-180.451200,-603.729100,88.350092,-0.177617,0.005730
C03233=2039.536800,-180.466700,-603.729100,88.350092,-0.177617,0.005730
C03234=2126.724100,-180.496100,-603.729100,88.350092,-0.177617,0.005730
C03235=2071.360800,-180.520800,-603.729100,88.350092,-0.177617,0.005730
C03236=1870.091900,-180.550500,-603.729100,88.350092,-0.177617,0.005730
C03237=2032.672600,-180.579200,-603.729100,88.350092,-0.177617,0.005730
C03238=1861.018100,-180.602200,-603.729100,88.350092,-0.177617,0.005730
C03239=1856.342000,-180.627900,-603.729100,88.350092,-0.177617,0.005730
C03240=1962.636500,-180.654900,-603.729100,88.350092,-0.177617,0.005730
C03241=2045.705000,-180.685000,-603.729100,88.350092,-0.177617,0.005730
C03242=1879.519200,-180.738700,-603.729100,88.350092,-0.177617,0.005730
C03243=2003.485200,-180.788700,-603.729100,88.350092,-0.177617,0.005730
C03244=2098.169100,-180.820800,-603.729100,88.350092,-0.177617,0.005730
C03245=2143.097000,-180.856600,-603.729100,88.350092,-0.177617,0.005730
C03246=2104.493500,-180.919100,-603.729100,88.350092,-0.177617,0.005730
C03247=1846.729500,-180.981300,-603.729100,88.350092,-0.177617,0.005730
C03248=1846.317800,-181.066800,-603.729100,88.350092,-0.177617,0.005730
C03249=2142.794800,-181.099500,-603.729100,88.350092,-0.177617,0.005730
C03250=1841.155900,-181.191800,-603.729100,88.350092,-0.177617,0.005730
C03251=2134.639000,-181.220500,-603.729100,88.350092,-0.177617,0.005730
C03252=2141.629600,-181.318100,-603.729100,88.350092,-0.177617,0.005730
C03253=1839.002200,-181.339700,-603.729100,88.350092,-0.177617,0.005730
C03254=1835.088400,-181.393800,-603.729100,88.350092,-0.177617,0.005730
C03255=2159.626800,-181.495100,-603.729100,88.350092,-0.177617,0.005730
C03256=1831.981100,-181.566400,-603.729100,88.350092,-0.177617,0.005730
C03257=2155.251100,-181.633700,-603.729100,88.350092,-0.177617,0.005730
C03258=1826.691200,-181.767800,-603.729100,88.350092,-0.177617,0.005730
C03259=1821.509100,-181.853600,-603.729100,88.350092,-0.177617,0.005730
C03260=2167.914500,-181.899900,-603.729100,88.350092,-0.177617,0.005730
C03261=1818.626600,-182.031000,-603.729100,88.350092,-0.177617,0.005730
C03262=1820.438700,-182.096200,-603.729100,88.350092,-0.177617,0.005730
C03263=1814.338100,-182.192800,-603.729100,88.350092,-0.177617,0.005730
C03264=2175.374500,-182.266400,-603.729100,88.350092,-0.177617,0.005730
C03265=2171.130200,-182.310900,-603.729100,88.350092,-0.177617,0.005730
C03266=1807.574600,-182.368100,-603.729100,88.350092,-0.177617,0.005730
C03267=1810.938000,-182.424200,-603.729100,88.350092,-0.177617,0.005730
C03268=1810.029400,-182.466500,-603.729100,88.350092,-0.177617,0.005730
C03269=1804.802600,-182.526300,-603.729100,88.350092,-0.177617,0.005730
C03270=1797.703700,-182.641500,-603.729100,88.350092,-0.177617,0.005730
C03271=1794.623600,-182.685400,-603.729100,88.350092,-0.177617,0.005730
C03272=1798.581700,-182.699600,-603.729100,88.350092,-0.177617,0.005730
C03273=1801.296900,-182.864100,-603.729100,88.350092,-0.177617,0.005730
C03274=1794.173700,-182.912400,-603.729100,88.350092,-0.177617,0.005730
C03275=2186.248200,-182.984400,-603.729100,88.350092,-0.177617,0.005730
C03276=1796.027900,-183.101300,-603.729100,88.350092,-0.177617,0.005730
C03277=2189.399200,-183.207400,-603.729100,88.350092,-0.177617,0.005730
C03278=1795.576200,-183.328300,-603.729100,88.350092,-0.177617,0.005730
C03279=1797.530500,-183.798200,-653.729100,88.350092,-0.177617,0.005730
C03280=1794.807300,-183.543500,-653.729100,88.350092,-0.177617,0.005730
C03281=2189.771400,-183.334700,-653.729100,88.350092,-0.177617,0.005730
C03282=1802.266900,-183.224200,-653.729100,88.350092,-0.177617,0.005730
C03283=1802.037900,-183.126300,-653.729100,88.350092,-0.177617,0.005730
C03284=2185.631800,-183.055000,-653.729100,88.350092,-0.177617,0.005730
C03285=2192.211600,-182.994200,-653.729100,88.350092,-0.177617,0.005730
C03286=2185.781500,-182.916300,-653.729100,88.350092,-0.177617,0.005730
C03287=1802.817300,-182.773200,-653.729100,88.350092,-0.177617,0.005730
C03288=1810.043300,-182.701900,-653.729100,88.350092,-0.177617,0.005730
C03289=1809.242000,-182.593100,-653.729100,88.350092,-0.177617,0.005730
C03290=2176.026900,-182.439600,-653.729100,88.350092,-0.177617,0.005730
C03291=2176.069100,-182.326900,-653.729100,88.350092,-0.177617,0.005730
C03292=1819.775400,-182.197600,-653.729100,88.350092,-0.177617,0.005730
C03293=2170.601400,-182.081600,-653.729100,88.350092,-0.177617,0.005730
C03294=2169.427700,-182.035200,-653.729100,88.350092,-0.177617,0.005730
C03295=1826.625400,-181.825200,-653.729100,88.350092,-0.177617,0.005730
C03296=1830.658700,-181.646200,-653.729100,88.350092,-0.177617,0.005730
C03297=2162.606900,-181.498900,-653.729100,88.350092,-0.177617,0.005730
C03298=1835.342800,-181.367100,-653.729100,88.350092,-0.177617,0.005730
C03299=2155.475100,-181.264700,-653.729100,88.350092,-0.177617,0.005730
C03300=1841.387000,-181.129900,-653.729100,88.350092,-0.177617,0.005730
C03301=1834.901600,-181.089100,-653.729100,88.350092,-0.177617,0.005730
C03302=1844.405200,-180.890100,-653.729100,88.350092,-0.177617,0.005730
C03303=1848.633600,-180.790100,-653.729100,88.350092,-0.177617,0.005730
C03304=1852.411100,-180.728600,-653.729100,88.350092,-0.177617,0.005730
C03305=1845.659100,-180.627600,-653.729100,88.350092,-0.177617,0.005730
C03306=2140.455700,-180.574900,-653.729100,88.350092,-0.177617,0.005730
C03307=1855.524300,-180.450200,-653.729100,88.350092,-0.177617,0.005730
C03308=1860.187100,-180.338000,-653.729100,88.350092,-0.177617,0.005730
C03309=1858.387600,-180.263400,-653.729100,88.350092,-0.177617,0.005730
C03310=1870.391500,-180.154900,-653.729100,88.350092,-0.177617,0.005730
C03311=1864.238500,-180.096500,-653.729100,88.350092,-0.177617,0.005730
C03312=2121.275300,-180.061000,-653.729100,88.350092,-0.177617,0.005730
C03313=2116.445800,-179.991400,-653.729100,88.350092,-0.177617,0.005730
C03314=1869.570700,-179.959300,-653.729100,88.350092,-0.177617,0.005730
C03315=1874.753200,-179.895400,-653.729100,88.350092,-0.177617,0.005730
C03316=2115.274200,-179.842200,-653.729100,88.350092,-0.177617,0.005730
C03317=1883.706700,-179.763000,-653.729100,88.350092,-0.177617,0.005730
C03318=2113.231200,-179.694800,-653.729100,88.350092,-0.177617,0.005730
C03319=1871.170500,-179.630900,-653.729100,88.350092,-0.177617,0.005730
C03320=1880.695700,-179.580600,-653.729100,88.350092,-0.177617,0.005730
C03321=1894.412600,-179.545100,-653.729100,88.350092,-0.177617,0.005730
C03322=1887.982300,-179.493700,-653.729100,88.350092,-0.177617,0.005730
C03323=2100.923700,-179.464900,-653.729100,88.350092,-0.177617,0.005730
C03324=2100.502300,-179.440400,-653.729100,88.350092,-0.177617,0.005730
C03325=1898.496500,-179.400500,-653.729100,88.350092,-0.177617,0.005730
C03326=2102.255100,-179.357600,-653.729100,88.350092,-0.177617,0.005730
C03327=2080.753700,-179.325500,-653.729100,88.350092,-0.177617,0.005730
C03328=2074.575100,-179.285300,-653.729100,88.350092,-0.177617,0.005730
C03329=1909.263100,-179.263700,-653.729100,88.350092,-0.177617,0.005730
C03330=1915.660700,-179.250100,-653.729100,88.350092,-0.177617,0.005730
C03331=1939.278900,-179.237600,-653.729100,88.350092,-0.177617,0.005730
C03332=1960.487800,-179.222100,-653.729100,88.350092,-0.177617,0.005730
C03333=2088.968600,-179.204200,-653.729100,88.350092,-0.177617,0.005730
C03334=2071.505800,-179.187000,-653.729100,88.350092,-0.177617,0.005730
C03335=1909.259200,-179.172800,-653.729100,88.350092,-0.177617,0.005730
C03336=2021.723900,-179.155900,-653.729100,88.350092,-0.177617,0.005730
C03337=2082.715300,-179.137300,-653.729100,88.350092,-0.177617,0.005730
C03338=2010.783500,-179.120400,-653.729100,88.350092,-0.177617,0.005730
C03339=1935.071900,-179.113200,-653.729100,88.350092,-0.177617,0.005730
C03340=1918.436400,-179.091700,-653.729100,88.350092,-0.177617,0.005730
C03341=2000.671300,-179.080900,-653.729100,88.350092,-0.177617,0.005730
C03342=2016.960000,-179.064700,-653.729100,88.350092,-0.177617,0.005730
C03343=2063.397200,-179.054500,-653.729100,88.350092,-0.177617,0.005730
C03344=2080.485000,-179.042700,-653.729100,88.350092,-0.177617,0.005730
C03345=2035.770800,-179.033300,-653.729100,88.350092,-0.177617,0.005730
C03346=1992.287100,-179.022100,-653.729100,88.350092,-0.177617,0.005730
C03347=2000.482100,-179.017700,-653.729100,88.350092,-0.177617,0.005730
C03348=1929.348700,-179.011000,-653.729100,88.350092,-0.177617,0.005730
C03349=1899.549400,-179.001500,-653.729100,88.350092,-0.177617,0.005730
C03350=1936.270500,-178.992400,-653.729100,88.350092,-0.177617,0.005730
C03351=2081.915800,-178.984600,-653.729100,88.350092,-0.177617,0.005730
C03352=1965.970400,-178.978500,-653.729100,88.350092,-0.177617,0.005730
C03353=1923.907200,-178.973500,-653.729100,88.350092,-0.177617,0.005730
C03354=1957.207900,-178.957200,-653.729100,88.350092,-0.177617,0.005730
C03355=2035.993900,-178.950200,-653.729100,88.350092,-0.177617,0.005730
C03356=1897.947500,-178.938000,-653.729100,88.350092,-0.177617,0.005730
C03357=2023.982400,-178.922100,-653.729100,88.350092,-0.177617,0.005730
C03358=1973.587200,-178.908300,-653.729100,88.350092,-0.177617,0.005730
C03359=1913.597900,-178.881600,-653.729100,88.350092,-0.177617,0.005730
C03360=1971.203400,-178.871800,-653.729100,88.350092,-0.177617,0.005730
C03361=1957.762500,-178.855900,-653.729100,88.350092,-0.177617,0.005730
C03362=1949.669900,-178.842400,-653.729100,88.350092,-0.177617,0.005730
C03363=2008.811800,-178.834600,-653.729100,88.350092,-0.177617,0.005730
C03364=1927.055300,-178.826800,-653.729100,88.350092,-0.177617,0.005730
C03365=2028.238100,-178.817400,-653.729100,88.350092,-0.177617,0.005730
C03366=1952.212900,-178.807200,-653.729100,88.350092,-0.177617,0.005730
C03367=1940.350500,-178.790700,-653.729100,88.350092,-0.177617,0.005730
C03368=2018.917100,-178.776500,-653.729100,88.350092,-0.177617,0.005730
C03369=2042.360400,-178.763000,-653.729100,88.350092,-0.177617,0.005730
C03370=1951.895700,-178.740400,-653.729100,88.350092,-0.177617,0.005730
C03371=1972.852000,-178.719700,-653.729100,88.350092,-0.177617,0.005730
C03372=1963.973700,-178.702200,-653.729100,88.350092,-0.177617,0.005730
C03373=2004.466900,-178.669400,-653.729100,88.350092,-0.177617,0.005730
C03374=1966.162700,-178.647100,-653.729100,88.350092,-0.177617,0.005730
C03375=1945.662400,-178.470700,-703.729100,88.350092,-0.177617,0.005730
C03376=1997.752600,-178.539700,-703.729100,88.350092,-0.177617,0.005730
C03377=1947.426300,-178.563300,-703.729100,88.350092,-0.177617,0.005730
C03378=1941.006500,-178.594400,-703.729100,88.350092,-0.177617,0.005730
C03379=1954.269200,-178.606700,-703.729100,88.350092,-0.177617,0.005730
C03380=2007.056300,-178.619100,-703.729100,88.350092,-0.177617,0.005730
C03381=1983.653100,-178.630900,-703.729100,88.350092,-0.177617,0.005730
C03382=1920.468100,-178.647100,-703.729100,88.350092,-0.177617,0.005730
C03383=1932.254900,-178.658900,-703.729100,88.350092,-0.177617,0.005730
C03384=1927.071300,-178.673800,-703.729100,88.350092,-0.177617,0.005730
C03385=2013.934700,-178.689700,-703.729100,88.350092,-0.177617,0.005730
C03386=1970.871100,-178.696400,-703.729100,88.350092,-0.177617,0.005730
C03387=2011.917000,-178.703200,-703.729100,88.350092,-0.177617,0.005730
C03388=1941.197800,-178.712300,-703.729100,88.350092,-0.177617,0.005730
C03389=2028.948000,-178.726500,-703.729100,88.350092,-0.177617,0.005730
C03390=2021.823100,-178.733600,-703.729100,88.350092,-0.177617,0.005730
C03391=1992.015700,-178.739700,-703.729100,88.350092,-0.177617,0.005730
C03392=1912.673200,-178.745100,-703.729100,88.350092,-0.177617,0.005730
C03393=1956.205500,-178.750800,-703.729100,88.350092,-0.177617,0.005730
C03394=1913.789600,-178.756200,-703.729100,88.350092,-0.177617,0.005730
C03395=2033.677800,-178.762600,-703.729100,88.350092,-0.177617,0.005730
C03396=2040.992700,-178.770100,-703.729100,88.350092,-0.177617,0.005730
C03397=1958.929400,-178.792000,-703.729100,88.350092,-0.177617,0.005730
C03398=1911.327100,-178.813000,-703.729100,88.350092,-0.177617,0.005730
C03399=1919.115000,-178.822800,-703.729100,88.350092,-0.177617,0.005730
C03400=2048.021100,-178.828900,-703.729100,88.350092,-0.177617,0.005730
C03401=1907.755600,-178.848800,-703.729100,88.350092,-0.177617,0.005730
C03402=2034.024600,-178.866000,-703.729100,88.350092,-0.177617,0.005730
C03403=1903.842800,-178.878200,-703.729100,88.350092,-0.177617,0.005730
C03404=2029.183300,-178.889000,-703.729100,88.350092,-0.177617,0.005730
C03405=1888.802000,-178.910300,-703.729100,88.350092,-0.177617,0.005730
C03406=2023.997000,-178.936000,-703.729100,88.350092,-0.177617,0.005730
C03407=2039.685000,-178.959600,-703.729100,88.350092,-0.177617,0.005730
C03408=1983.435100,-178.976800,-703.729100,88.350092,-0.177617,0.005730
C03409=1896.739800,-178.989700,-703.729100,88.350092,-0.177617,0.005730
C03410=2064.780600,-179.001500,-703.729100,88.350092,-0.177617,0.005730
C03411=2072.676500,-179.026800,-703.729100,88.350092,-0.177617,0.005730
C03412=1886.765800,-179.057900,-703.729100,88.350092,-0.177617,0.005730
C03413=2061.175900,-179.087700,-703.729100,88.350092,-0.177617,0.005730
C03414=2044.467000,-179.117700,-703.729100,88.350092,-0.177617,0.005730
C03415=1887.896200,-179.146100,-703.729100,88.350092,-0.177617,0.005730
C03416=2030.542600,-179.165400,-703.729100,88.350092,-0.177617,0.005730
C03417=2050.832800,-179.196400,-703.729100,88.350092,-0.177617,0.005730
C03418=2081.592000,-179.231900,-703.729100,88.350092,-0.177617,0.005730
C03419=2090.908600,-179.276900,-703.729100,88.350092,-0.177617,0.005730
C03420=1883.035400,-179.314400,-703.729100,88.350092,-0.177617,0.005730
C03421=1867.904300,-179.363000,-703.729100,88.350092,-0.177617,0.005730
C03422=1867.211700,-179.387000,-703.729100,88.350092,-0.177617,0.005730
C03423=2057.321400,-179.413300,-703.729100,88.350092,-0.177617,0.005730
C03424=1861.517200,-179.484600,-703.729100,88.350092,-0.177617,0.005730
C03425=2088.727100,-179.535000,-703.729100,88.350092,-0.177617,0.005730
C03426=2068.367100,-179.583400,-703.729100,88.350092,-0.177617,0.005730
C03427=1868.992800,-179.656900,-703.729100,88.350092,-0.177617,0.005730
C03428=2087.980800,-179.724500,-703.729100,88.350092,-0.177617,0.005730
C03429=2094.776800,-179.777500,-703.729100,88.350092,-0.177617,0.005730
C03430=1848.981400,-179.859600,-703.729100,88.350092,-0.177617,0.005730
C03431=1850.535200,-179.978900,-703.729100,88.350092,-0.177617,0.005730
C03432=2119.439100,-180.044800,-703.729100,88.350092,-0.177617,0.005730
C03433=1844.904800,-180.139400,-703.729100,88.350092,-0.177617,0.005730
C03434=1841.705900,-180.159300,-703.729100,88.350092,-0.177617,0.005730
C03435=1844.310600,-180.269100,-703.729100,88.350092,-0.177617,0.005730
C03436=2126.819600,-180.342400,-703.729100,88.350092,-0.177617,0.005730
C03437=1832.434200,-180.372100,-703.729100,88.350092,-0.177617,0.005730
C03438=2132.367400,-180.549200,-703.729100,88.350092,-0.177617,0.005730
C03439=1836.658600,-180.617800,-703.729100,88.350092,-0.177617,0.005730
C03440=2116.198000,-180.698200,-703.729100,88.350092,-0.177617,0.005730
C03441=2122.359600,-180.784000,-703.729100,88.350092,-0.177617,0.005730
C03442=2134.332800,-180.928900,-703.729100,88.350092,-0.177617,0.005730
C03443=1820.555100,-181.032000,-703.729100,88.350092,-0.177617,0.005730
C03444=1825.968000,-181.189100,-703.729100,88.350092,-0.177617,0.005730
C03445=2145.016800,-181.239700,-703.729100,88.350092,-0.177617,0.005730
C03446=1815.870600,-181.356000,-703.729100,88.350092,-0.177617,0.005730
C03447=1814.977300,-181.424900,-703.729100,88.350092,-0.177617,0.005730
C03448=1827.581400,-181.469500,-703.729100,88.350092,-0.177617,0.005730
C03449=1810.984400,-181.765400,-703.729100,88.350092,-0.177617,0.005730
C03450=1803.869900,-181.839100,-703.729100,88.350092,-0.177617,0.005730
C03451=2153.754800,-181.865100,-703.729100,88.350092,-0.177617,0.005730
C03452=1800.030700,-182.006400,-703.729100,88.350092,-0.177617,0.005730
C03453=2160.483900,-182.162100,-703.729100,88.350092,-0.177617,0.005730
C03454=2171.893100,-182.251200,-703.729100,88.350092,-0.177617,0.005730
C03455=1792.127200,-182.359500,-703.729100,88.350092,-0.177617,0.005730
C03456=1796.827800,-182.483300,-703.729100,88.350092,-0.177617,0.005730
C03457=2175.948100,-182.581000,-703.729100,88.350092,-0.177617,0.005730
C03458=2172.656100,-182.725600,-703.729100,88.350092,-0.177617,0.005730
C03459=1804.373200,-182.814800,-703.729100,88.350092,-0.177617,0.005730
C03460=1793.756500,-182.955700,-703.729100,88.350092,-0.177617,0.005730
C03461=1792.095600,-183.141500,-703.729100,88.350092,-0.177617,0.005730
C03462=2182.167200,-183.277300,-703.729100,88.350092,-0.177617,0.005730
C03463=2185.395900,-183.508100,-703.729100,88.350092,-0.177617,0.005730
C03464=2189.609300,-183.716300,-703.729100,88.350092,-0.177617,0.005730
C03465=2190.764800,-184.054300,-753.729100,88.350092,-0.177617,0.005730
C03466=2184.710200,-183.884400,-753.729100,88.350092,-0.177617,0.005730
C03467=2180.199700,-183.783400,-753.729100,88.350092,-0.177617,0.005730
C03468=2186.600400,-183.693500,-753.729100,88.350092,-0.177617,0.005730
C03469=2191.846700,-183.586800,-753.729100,88.350092,-0.177617,0.005730
C03470=2167.598400,-183.490500,-753.729100,88.350092,-0.177617,0.005730
C03471=2172.853400,-183.355700,-753.729100,88.350092,-0.177617,0.005730
C03472=2164.129300,-183.133400,-753.729100,88.350092,-0.177617,0.005730
C03473=2170.563100,-183.037100,-753.729100,88.350092,-0.177617,0.005730
C03474=2146.473000,-182.795500,-753.729100,88.350092,-0.177617,0.005730
C03475=2166.801600,-182.657000,-753.729100,88.350092,-0.177617,0.005730
C03476=2152.832600,-182.455600,-753.729100,88.350092,-0.177617,0.005730
C03477=1791.225400,-182.386000,-753.729100,88.350092,-0.177617,0.005730
C03478=2154.422000,-182.204300,-753.729100,88.350092,-0.177617,0.005730
C03479=1794.686500,-182.090100,-753.729100,88.350092,-0.177617,0.005730
C03480=2122.317100,-181.996800,-753.729100,88.350092,-0.177617,0.005730
C03481=2116.270500,-181.874900,-753.729100,88.350092,-0.177617,0.005730
C03482=1799.750400,-181.794500,-753.729100,88.350092,-0.177617,0.005730
C03483=1799.939900,-181.676200,-753.729100,88.350092,-0.177617,0.005730
C03484=2100.157600,-181.610700,-753.729100,88.350092,-0.177617,0.005730
C03485=2131.464700,-181.519800,-753.729100,88.350092,-0.177617,0.005730
C03486=1812.286500,-181.468100,-753.729100,88.350092,-0.177617,0.005730
C03487=1807.445900,-181.372200,-753.729100,88.350092,-0.177617,0.005730
C03488=2102.146100,-181.288000,-753.729100,88.350092,-0.177617,0.005730
C03489=2085.435400,-181.179300,-753.729100,88.350092,-0.177617,0.005730
C03490=2078.922800,-181.095800,-753.729100,88.350092,-0.177617,0.005730
C03491=2125.468600,-181.067400,-753.729100,88.350092,-0.177617,0.005730
C03492=2075.192300,-180.986000,-753.729100,88.350092,-0.177617,0.005730
C03493=2110.263700,-180.884300,-753.729100,88.350092,-0.177617,0.005730
C03494=1818.147000,-180.811000,-753.729100,88.350092,-0.177617,0.005730
C03495=2085.562300,-180.739000,-753.729100,88.350092,-0.177617,0.005730
C03496=1828.269100,-180.684000,-753.729100,88.350092,-0.177617,0.005730
C03497=2088.248500,-180.625500,-753.729100,88.350092,-0.177617,0.005730
C03498=2049.037500,-180.489500,-753.729100,88.350092,-0.177617,0.005730
C03499=2019.267400,-180.448800,-753.729100,88.350092,-0.177617,0.005730
C03500=2080.518800,-180.416100,-753.729100,88.350092,-0.177617,0.005730
C03501=2034.341800,-180.377900,-753.729100,88.350092,-0.177617,0.005730
C03502=1830.157200,-180.357300,-753.729100,88.350092,-0.177617,0.005730
C03503=1828.212300,-180.315400,-753.729100,88.350092,-0.177617,0.005730
C03504=2083.945000,-180.245800,-753.729100,88.350092,-0.177617,0.005730
C03505=1833.544300,-180.205300,-753.729100,88.350092,-0.177617,0.005730
C03506=2028.700700,-180.164000,-753.729100,88.350092,-0.177617,0.005730
C03507=1838.876700,-180.102900,-753.729100,88.350092,-0.177617,0.005730
C03508=2015.079100,-180.063000,-753.729100,88.350092,-0.177617,0.005730
C03509=2018.684100,-180.036000,-753.729100,88.350092,-0.177617,0.005730
C03510=2077.341500,-179.965700,-753.729100,88.350092,-0.177617,0.005730
C03511=1844.604500,-179.898800,-753.729100,88.350092,-0.177617,0.005730
C03512=2048.595900,-179.880200,-753.729100,88.350092,-0.177617,0.005730
C03513=2014.904100,-179.826200,-753.729100,88.350092,-0.177617,0.005730
C03514=2074.182600,-179.788300,-753.729100,88.350092,-0.177617,0.005730
C03515=1958.379700,-179.769800,-753.729100,88.350092,-0.177617,0.005730
C03516=1849.029200,-179.729900,-753.729100,88.350092,-0.177617,0.005730
C03517=1914.456400,-179.708300,-753.729100,88.350092,-0.177617,0.005730
C03518=1971.224100,-179.680600,-753.729100,88.350092,-0.177617,0.005730
C03519=2052.805600,-179.655900,-753.729100,88.350092,-0.177617,0.005730
C03520=2018.762000,-179.632600,-753.729100,88.350092,-0.177617,0.005730
C03521=2013.584400,-179.607300,-753.729100,88.350092,-0.177617,0.005730
C03522=2028.413200,-179.576900,-753.729100,88.350092,-0.177617,0.005730
C03523=2055.918100,-179.559000,-753.729100,88.350092,-0.177617,0.005730
C03524=1909.610900,-179.527500,-753.729100,88.350092,-0.177617,0.005730
C03525=1935.151600,-179.516000,-753.729100,88.350092,-0.177617,0.005730
C03526=1857.146100,-179.504600,-753.729100,88.350092,-0.177617,0.005730
C03527=1931.535800,-179.476900,-753.729100,88.350092,-0.177617,0.005730
C03528=1904.805900,-179.440400,-753.729100,88.350092,-0.177617,0.005730
C03529=1917.259700,-179.428900,-753.729100,88.350092,-0.177617,0.005730
C03530=1978.561300,-179.401900,-753.729100,88.350092,-0.177617,0.005730
C03531=1869.525700,-179.389200,-753.729100,88.350092,-0.177617,0.005730
C03532=1961.877100,-179.367700,-753.729100,88.350092,-0.177617,0.005730
C03533=2028.982900,-179.348100,-753.729100,88.350092,-0.177617,0.005730
C03534=1872.671000,-179.328200,-753.729100,88.350092,-0.177617,0.005730
C03535=1936.671300,-179.300500,-753.729100,88.350092,-0.177617,0.005730
C03536=2033.710500,-179.279600,-753.729100,88.350092,-0.177617,0.005730
C03537=1903.326600,-179.268400,-753.729100,88.350092,-0.177617,0.005730
C03538=1867.151400,-179.247500,-753.729100,88.350092,-0.177617,0.005730
C03539=1874.034900,-179.231900,-753.729100,88.350092,-0.177617,0.005730
C03540=1878.333800,-179.215400,-753.729100,88.350092,-0.177617,0.005730
C03541=1944.501700,-179.198100,-753.729100,88.350092,-0.177617,0.005730
C03542=1905.223800,-179.187300,-753.729100,88.350092,-0.177617,0.005730
C03543=2005.268100,-179.150800,-753.729100,88.350092,-0.177617,0.005730
C03544=1878.784800,-179.120400,-753.729100,88.350092,-0.177617,0.005730
C03545=1885.658500,-179.081600,-753.729100,88.350092,-0.177617,0.005730
C03546=1954.477800,-179.053900,-753.729100,88.350092,-0.177617,0.005730
C03547=1907.170000,-179.039000,-753.729100,88.350092,-0.177617,0.005730
C03548=1973.983500,-179.008300,-753.729100,88.350092,-0.177617,0.005730
C03549=1990.414300,-178.979900,-753.729100,88.350092,-0.177617,0.005730
C03550=1977.276800,-178.948800,-753.729100,88.350092,-0.177617,0.005730
C03551=1911.571100,-178.934300,-753.729100,88.350092,-0.177617,0.005730
C03552=1903.480000,-178.905900,-753.729100,88.350092,-0.177617,0.005730
C03553=1927.658200,-178.819400,-753.729100,88.350092,-0.177617,0.005730
C03554=1910.732500,-179.518700,-803.729100,88.350092,-0.177617,0.005730
C03555=1924.471800,-179.616000,-803.729100,88.350092,-0.177617,0.005730
C03556=1920.740300,-179.693100,-803.729100,88.350092,-0.177617,0.005730
C03557=1903.865500,-179.747100,-803.729100,88.350092,-0.177617,0.005730
C03558=1899.964900,-179.796500,-803.729100,88.350092,-0.177617,0.005730
C03559=1897.454700,-179.873100,-803.729100,88.350092,-0.177617,0.005730
C03560=1910.833800,-179.898500,-803.729100,88.350092,-0.177617,0.005730
C03561=1861.378800,-179.924200,-803.729100,88.350092,-0.177617,0.005730
C03562=1930.898000,-179.960000,-803.729100,88.350092,-0.177617,0.005730
C03563=1855.199800,-179.991700,-803.729100,88.350092,-0.177617,0.005730
C03564=1894.463800,-180.027900,-803.729100,88.350092,-0.177617,0.005730
C03565=1861.322400,-180.057300,-803.729100,88.350092,-0.177617,0.005730
C03566=1851.358800,-180.080600,-803.729100,88.350092,-0.177617,0.005730
C03567=1948.870400,-180.123200,-803.729100,88.350092,-0.177617,0.005730
C03568=1885.006700,-180.170800,-803.729100,88.350092,-0.177617,0.005730
C03569=1921.302500,-180.210300,-803.729100,88.350092,-0.177617,0.005730
C03570=1962.425800,-180.276200,-803.729100,88.350092,-0.177617,0.005730
C03571=1914.681500,-180.301500,-803.729100,88.350092,-0.177617,0.005730
C03572=1968.159000,-180.349800,-803.729100,88.350092,-0.177617,0.005730
C03573=1935.978400,-180.363400,-803.729100,88.350092,-0.177617,0.005730
C03574=1861.583400,-180.394400,-803.729100,88.350092,-0.177617,0.005730
C03575=1939.074200,-180.409300,-803.729100,88.350092,-0.177617,0.005730
C03576=1828.435000,-180.433600,-803.729100,88.350092,-0.177617,0.005730
C03577=1971.285800,-180.468400,-803.729100,88.350092,-0.177617,0.005730
C03578=2024.581200,-180.493400,-803.729100,88.350092,-0.177617,0.005730
C03579=1893.315000,-180.538400,-803.729100,88.350092,-0.177617,0.005730
C03580=1960.993000,-180.565100,-803.729100,88.350092,-0.177617,0.005730
C03581=1833.742000,-180.585300,-803.729100,88.350092,-0.177617,0.005730
C03582=1849.660000,-180.627600,-803.729100,88.350092,-0.177617,0.005730
C03583=1975.490800,-180.646100,-803.729100,88.350092,-0.177617,0.005730
C03584=1826.428800,-180.667800,-803.729100,88.350092,-0.177617,0.005730
C03585=2006.352500,-180.697200,-803.729100,88.350092,-0.177617,0.005730
C03586=1852.293300,-180.722800,-803.729100,88.350092,-0.177617,0.005730
C03587=1888.721500,-180.765100,-803.729100,88.350092,-0.177617,0.005730
C03588=1976.461300,-180.795800,-803.729100,88.350092,-0.177617,0.005730
C03589=1919.247800,-180.815700,-803.729100,88.350092,-0.177617,0.005730
C03590=2034.664200,-180.846500,-803.729100,88.350092,-0.177617,0.005730
C03591=1940.495900,-180.871500,-803.729100,88.350092,-0.177617,0.005730
C03592=1817.552700,-180.896800,-803.729100,88.350092,-0.177617,0.005730
C03593=2040.840400,-180.947700,-803.729100,88.350092,-0.177617,0.005730
C03594=1987.402000,-180.967400,-803.729100,88.350092,-0.177617,0.005730
C03595=1821.487400,-181.000900,-803.729100,88.350092,-0.177617,0.005730
C03596=1930.308600,-181.022500,-803.729100,88.350092,-0.177617,0.005730
C03597=2027.560900,-181.041800,-803.729100,88.350092,-0.177617,0.005730
C03598=1948.775200,-181.057600,-803.729100,88.350092,-0.177617,0.005730
C03599=2039.090000,-181.094100,-803.729100,88.350092,-0.177617,0.005730
C03600=2074.779300,-181.139400,-803.729100,88.350092,-0.177617,0.005730
C03601=1825.388700,-181.151900,-803.729100,88.350092,-0.177617,0.005730
C03602=2023.232700,-181.185300,-803.729100,88.350092,-0.177617,0.005730
C03603=1808.970000,-181.241400,-803.729100,88.350092,-0.177617,0.005730
C03604=1815.914500,-181.273900,-803.729100,88.350092,-0.177617,0.005730
C03605=2006.035000,-181.312700,-803.729100,88.350092,-0.177617,0.005730
C03606=2050.567600,-181.372800,-803.729100,88.350092,-0.177617,0.005730
C03607=2018.328900,-181.434000,-803.729100,88.350092,-0.177617,0.005730
C03608=1807.799400,-181.463700,-803.729100,88.350092,-0.177617,0.005730
C03609=2061.572600,-181.542400,-803.729100,88.350092,-0.177617,0.005730
C03610=1809.892000,-181.572200,-803.729100,88.350092,-0.177617,0.005730
C03611=2080.950300,-181.596500,-803.729100,88.350092,-0.177617,0.005730
C03612=2014.492600,-181.642100,-803.729100,88.350092,-0.177617,0.005730
C03613=1800.297600,-181.701600,-803.729100,88.350092,-0.177617,0.005730
C03614=1800.067400,-181.738900,-803.729100,88.350092,-0.177617,0.005730
C03615=2084.722300,-181.786700,-803.729100,88.350092,-0.177617,0.005730
C03616=2081.679100,-181.854600,-803.729100,88.350092,-0.177617,0.005730
C03617=1804.542900,-181.901600,-803.729100,88.350092,-0.177617,0.005730
C03618=2061.315300,-181.946200,-803.729100,88.350092,-0.177617,0.005730
C03619=2111.251800,-182.005000,-803.729100,88.350092,-0.177617,0.005730
C03620=2058.575800,-182.029300,-803.729100,88.350092,-0.177617,0.005730
C03621=1794.344900,-182.075900,-803.729100,88.350092,-0.177617,0.005730
C03622=2064.982000,-182.118100,-803.729100,88.350092,-0.177617,0.005730
C03623=2102.867200,-182.186400,-803.729100,88.350092,-0.177617,0.005730
C03624=2089.390700,-182.230000,-803.729100,88.350092,-0.177617,0.005730
C03625=2080.350300,-182.313900,-803.729100,88.350092,-0.177617,0.005730
C03626=2086.042600,-182.353300,-803.729100,88.350092,-0.177617,0.005730
C03627=2091.647500,-182.421900,-803.729100,88.350092,-0.177617,0.005730
C03628=2080.244500,-182.656300,-803.729100,88.350092,-0.177617,0.005730
C03629=2091.809900,-182.836400,-803.729100,88.350092,-0.177617,0.005730
C03630=2115.868600,-182.973200,-803.729100,88.350092,-0.177617,0.005730
C03631=2116.908700,-183.067100,-803.729100,88.350092,-0.177617,0.005730
C03632=2129.241600,-183.171500,-803.729100,88.350092,-0.177617,0.005730
C03633=2135.314000,-183.362100,-803.729100,88.350092,-0.177617,0.005730
C03634=2128.051700,-183.455000,-803.729100,88.350092,-0.177617,0.005730
C03635=2140.242100,-183.548600,-803.729100,88.350092,-0.177617,0.005730
C03636=2133.355200,-183.704300,-803.729100,88.350092,-0.177617,0.005730
C03637=2152.621700,-183.786400,-803.729100,88.350092,-0.177617,0.005730
C03638=2139.611900,-183.942500,-803.729100,88.350092,-0.177617,0.005730
C03639=2177.275400,-183.974300,-803.729100,88.350092,-0.177617,0.005730
C03640=2174.109900,-184.096600,-803.729100,88.350092,-0.177617,0.005730
C03641=2184.252400,-184.158900,-803.729100,88.350092,-0.177617,0.005730
C03642=2154.457500,-184.255700,-803.729100,88.350092,-0.177617,0.005730
C03643=2180.306300,-184.309200,-803.729100,88.350092,-0.177617,0.005730
C03644=2191.291100,-184.376300,-803.729100,88.350092,-0.177617,0.005730
C03645=2176.588800,-184.449300,-803.729100,88.350092,-0.177617,0.005730
C03646=2177.846700,-184.559400,-803.729100,88.350092,-0.177617,0.005730
C03647=2189.316800,-184.923400,-853.729100,88.350092,-0.177617,0.005730
C03648=2183.704700,-184.853300,-853.729100,88.350092,-0.177617,0.005730
C03649=2181.051900,-184.741500,-853.729100,88.350092,-0.177617,0.005730
C03650=2185.083500,-184.707400,-853.729100,88.350092,-0.177617,0.005730
C03651=2175.979800,-184.675300,-853.729100,88.350092,-0.177617,0.005730
C03652=2186.097800,-184.642500,-853.729100,88.350092,-0.177617,0.005730
C03653=2173.145800,-184.590800,-853.729100,88.350092,-0.177617,0.005730
C03654=2159.100100,-184.536400,-853.729100,88.350092,-0.177617,0.005730
C03655=2169.010300,-184.503300,-853.729100,88.350092,-0.177617,0.005730
C03656=2161.607600,-184.495600,-853.729100,88.350092,-0.177617,0.005730
C03657=2190.500300,-184.441500,-853.729100,88.350092,-0.177617,0.005730
C03658=2150.847300,-184.410800,-853.729100,88.350092,-0.177617,0.005730
C03659=2154.428200,-184.350600,-853.729100,88.350092,-0.177617,0.005730
C03660=2154.393400,-184.274900,-853.729100,88.350092,-0.177617,0.005730
C03661=2142.222200,-184.227300,-853.729100,88.350092,-0.177617,0.005730
C03662=2129.510700,-184.132400,-853.729100,88.350092,-0.177617,0.005730
C03663=2126.214500,-184.029700,-853.729100,88.350092,-0.177617,0.005730
C03664=2122.824900,-183.939500,-853.729100,88.350092,-0.177617,0.005730
C03665=2135.909000,-183.824300,-853.729100,88.350092,-0.177617,0.005730
C03666=2105.186400,-183.761800,-853.729100,88.350092,-0.177617,0.005730
C03667=2126.722900,-183.702600,-853.729100,88.350092,-0.177617,0.005730
C03668=2094.309000,-183.649600,-853.729100,88.350092,-0.177617,0.005730
C03669=2063.453300,-183.571500,-853.729100,88.350092,-0.177617,0.005730
C03670=2075.227500,-183.481000,-853.729100,88.350092,-0.177617,0.005730
C03671=2098.062800,-183.411400,-853.729100,88.350092,-0.177617,0.005730
C03672=2065.427100,-183.300300,-853.729100,88.350092,-0.177617,0.005730
C03673=2099.168100,-183.252300,-853.729100,88.350092,-0.177617,0.005730
C03674=2092.393700,-183.208000,-853.729100,88.350092,-0.177617,0.005730
C03675=2071.759200,-183.154600,-853.729100,88.350092,-0.177617,0.005730
C03676=2093.931900,-183.087800,-853.729100,88.350092,-0.177617,0.005730
C03677=2043.097900,-183.029600,-853.729100,88.350092,-0.177617,0.005730
C03678=1792.952400,-183.005000,-853.729100,88.350092,-0.177617,0.005730
C03679=2029.748300,-182.936100,-853.729100,88.350092,-0.177617,0.005730
C03680=2064.124300,-182.890100,-853.729100,88.350092,-0.177617,0.005730
C03681=1794.338900,-182.854600,-853.729100,88.350092,-0.177617,0.005730
C03682=1806.096000,-182.816100,-853.729100,88.350092,-0.177617,0.005730
C03683=2013.750300,-182.796500,-853.729100,88.350092,-0.177617,0.005730
C03684=1831.355100,-182.769500,-853.729100,88.350092,-0.177617,0.005730
C03685=2039.176100,-182.734000,-853.729100,88.350092,-0.177617,0.005730
C03686=2003.431800,-182.688400,-853.729100,88.350092,-0.177617,0.005730
C03687=2025.813600,-182.665100,-853.729100,88.350092,-0.177617,0.005730
C03688=1816.366600,-182.639400,-853.729100,88.350092,-0.177617,0.005730
C03689=1977.868600,-182.629300,-853.729100,88.350092,-0.177617,0.005730
C03690=2004.050900,-182.593100,-853.729100,88.350092,-0.177617,0.005730
C03691=1901.935600,-182.573200,-853.729100,88.350092,-0.177617,0.005730
C03692=2052.170900,-182.544200,-853.729100,88.350092,-0.177617,0.005730
C03693=1804.499200,-182.529800,-853.729100,88.350092,-0.177617,0.005730
C03694=1839.522600,-182.513400,-853.729100,88.350092,-0.177617,0.005730
C03695=2020.243000,-182.500600,-853.729100,88.350092,-0.177617,0.005730
C03696=2040.170800,-182.483700,-853.729100,88.350092,-0.177617,0.005730
C03697=1977.011200,-182.463400,-853.729100,88.350092,-0.177617,0.005730
C03698=1957.970500,-182.456700,-853.729100,88.350092,-0.177617,0.005730
C03699=1914.038100,-182.440400,-853.729100,88.350092,-0.177617,0.005730
C03700=2017.243000,-182.425200,-853.729100,88.350092,-0.177617,0.005730
C03701=1815.955300,-182.390100,-853.729100,88.350092,-0.177617,0.005730
C03702=1932.650800,-182.377600,-853.729100,88.350092,-0.177617,0.005730
C03703=1962.626000,-182.361700,-853.729100,88.350092,-0.177617,0.005730
C03704=1995.024700,-182.345500,-853.729100,88.350092,-0.177617,0.005730
C03705=2035.249000,-182.321500,-853.729100,88.350092,-0.177617,0.005730
C03706=1894.181800,-182.296200,-853.729100,88.350092,-0.177617,0.005730
C03707=1865.165100,-182.253900,-853.729100,88.350092,-0.177617,0.005730
C03708=1821.895200,-182.233000,-853.729100,88.350092,-0.177617,0.005730
C03709=1896.381200,-182.221200,-853.729100,88.350092,-0.177617,0.005730
C03710=1813.401900,-182.208700,-853.729100,88.350092,-0.177617,0.005730
C03711=1907.311500,-182.191400,-853.729100,88.350092,-0.177617,0.005730
C03712=1916.412800,-182.173200,-853.729100,88.350092,-0.177617,0.005730
C03713=2050.538000,-182.145200,-853.729100,88.350092,-0.177617,0.005730
C03714=2012.001800,-182.119100,-853.729100,88.350092,-0.177617,0.005730
C03715=1840.669300,-182.087700,-853.729100,88.350092,-0.177617,0.005730
C03716=1972.814900,-182.061000,-853.729100,88.350092,-0.177617,0.005730
C03717=1808.740400,-182.020800,-853.729100,88.350092,-0.177617,0.005730
C03718=1878.622400,-181.974900,-853.729100,88.350092,-0.177617,0.005730
C03719=1884.691800,-181.963200,-853.729100,88.350092,-0.177617,0.005730
C03720=1859.525300,-181.952600,-853.729100,88.350092,-0.177617,0.005730
C03721=1827.761300,-181.922500,-853.729100,88.350092,-0.177617,0.005730
C03722=2014.040200,-181.902300,-853.729100,88.350092,-0.177617,0.005730
C03723=1959.314900,-181.849200,-853.729100,88.350092,-0.177617,0.005730
C03724=1998.634200,-181.825200,-853.729100,88.350092,-0.177617,0.005730
C03725=1922.193000,-181.811000,-853.729100,88.350092,-0.177617,0.005730
C03726=1997.691300,-181.758000,-853.729100,88.350092,-0.177617,0.005730
C03727=1954.492800,-181.728400,-853.729100,88.350092,-0.177617,0.005730
C03728=1858.833400,-181.697900,-853.729100,88.350092,-0.177617,0.005730
C03729=1825.171200,-181.678600,-853.729100,88.350092,-0.177617,0.005730
C03730=1855.433300,-181.620800,-853.729100,88.350092,-0.177617,0.005730
C03731=1979.753400,-181.574200,-853.729100,88.350092,-0.177617,0.005730
C03732=1835.829000,-181.531600,-853.729100,88.350092,-0.177617,0.005730
C03733=1895.720100,-181.508500,-853.729100,88.350092,-0.177617,0.005730
C03734=1842.560900,-181.462700,-853.729100,88.350092,-0.177617,0.005730
C03735=1924.486800,-181.413700,-853.729100,88.350092,-0.177617,0.005730
C03736=1921.588700,-181.364700,-853.729100,88.350092,-0.177617,0.005730
C03737=1847.603300,-181.337400,-853.729100,88.350092,-0.177617,0.005730
C03738=1894.768400,-181.285000,-853.729100,88.350092,-0.177617,0.005730
C03739=1903.645500,-181.249500,-853.729100,88.350092,-0.177617,0.005730
C03740=1910.157100,-181.170800,-853.729100,88.350092,-0.177617,0.005730
C03741=1850.415000,-181.076600,-853.729100,88.350092,-0.177617,0.005730
C03742=1863.131300,-180.990700,-853.729100,88.350092,-0.177617,0.005730
C03743=2216.165700,-99.670900,-454.076700,-102.863113,89.312661,167.137518
C03744=2214.487400,86.366300,-454.076700,-102.863113,89.312661,167.137518
C03745=2214.426100,214.921800,-454.076700,-102.863113,89.312661,167.137518
C03746=2213.771500,233.297600,-504.076700,-102.863113,89.312661,167.137518
C03747=2214.223900,229.665800,-504.076700,-102.863113,89.312661,167.137518
C03748=2213.605800,226.728900,-504.076700,-102.863113,89.312661,167.137518
C03749=2213.776700,225.236300,-504.076700,-102.863113,89.312661,167.137518
C03750=2213.620200,222.118600,-504.076700,-102.863113,89.312661,167.137518
C03751=2213.260500,218.869900,-504.076700,-102.863113,89.312661,167.137518
C03752=2213.705300,216.426900,-504.076700,-102.863113,89.312661,167.137518
C03753=2213.523900,212.165000,-504.076700,-102.863113,89.312661,167.137518
C03754=2213.573900,209.710200,-504.076700,-102.863113,89.312661,167.137518
C03755=2213.577400,205.553000,-504.076700,-102.863113,89.312661,167.137518
C03756=2213.781300,202.872600,-504.076700,-102.863113,89.312661,167.137518
C03757=2213.975700,197.022100,-504.076700,-102.863113,89.312661,167.137518
C03758=2213.913000,194.158500,-504.076700,-102.863113,89.312661,167.137518
C03759=2213.708600,191.004000,-504.076700,-102.863113,89.312661,167.137518
C03760=2213.526800,185.015400,-504.076700,-102.863113,89.312661,167.137518
C03761=2213.855100,179.768600,-504.076700,-102.863113,89.312661,167.137518
C03762=2213.597600,177.928200,-504.076700,-102.863113,89.312661,167.137518
C03763=2213.735200,173.041100,-504.076700,-102.863113,89.312661,167.137518
C03764=2214.250600,171.092100,-504.076700,-102.863113,89.312661,167.137518
C03765=2213.893100,168.011200,-504.076700,-102.863113,89.312661,167.137518
C03766=2213.927300,165.010500,-504.076700,-102.863113,89.312661,167.137518
C03767=2214.028400,162.003000,-504.076700,-102.863113,89.312661,167.137518
C03768=2213.813700,160.109000,-504.076700,-102.863113,89.312661,167.137518
C03769=2213.943000,156.746100,-504.076700,-102.863113,89.312661,167.137518
C03770=2214.247100,153.137700,-504.076700,-102.863113,89.312661,167.137518
C03771=2214.516300,148.218200,-504.076700,-102.863113,89.312661,167.137518
C03772=2214.565500,145.534300,-504.076700,-102.863113,89.312661,167.137518
C03773=2214.481600,141.873800,-504.076700,-102.863113,89.312661,167.137518
C03774=2214.302000,138.861500,-504.076700,-102.863113,89.312661,167.137518
C03775=2214.347600,136.153700,-504.076700,-102.863113,89.312661,167.137518
C03776=2214.021700,133.588800,-504.076700,-102.863113,89.312661,167.137518
C03777=2214.931100,130.308600,-504.076700,-102.863113,89.312661,167.137518
C03778=2214.461800,126.527600,-504.076700,-102.863113,89.312661,167.137518
C03779=2215.135000,123.766600,-504.076700,-102.863113,89.312661,167.137518
C03780=2214.075900,121.616900,-504.076700,-102.863113,89.312661,167.137518
C03781=2214.163100,118.315000,-504.076700,-102.863113,89.312661,167.137518
C03782=2214.060800,115.014000,-504.076700,-102.863113,89.312661,167.137518
C03783=2214.969800,112.614600,-504.076700,-102.863113,89.312661,167.137518
C03784=2214.711900,110.505100,-504.076700,-102.863113,89.312661,167.137518
C03785=2214.915400,106.124300,-504.076700,-102.863113,89.312661,167.137518
C03786=2215.225600,104.405600,-504.076700,-102.863113,89.312661,167.137518
C03787=2215.072800,101.798000,-504.076700,-102.863113,89.312661,167.137518
C03788=2214.430400,97.856500,-504.076700,-102.863113,89.312661,167.137518
C03789=2215.122500,96.432800,-504.076700,-102.863113,89.312661,167.137518
C03790=2214.461800,92.060300,-504.076700,-102.863113,89.312661,167.137518
C03791=2215.163600,90.117500,-504.076700,-102.863113,89.312661,167.137518
C03792=2214.700400,86.621800,-504.076700,-102.863113,89.312661,167.137518
C03793=2215.285900,82.970000,-504.076700,-102.863113,89.312661,167.137518
C03794=2215.585300,81.640800,-504.076700,-102.863113,89.312661,167.137518
C03795=2215.016800,77.326300,-504.076700,-102.863113,89.312661,167.137518
C03796=2216.113400,75.736000,-504.076700,-102.863113,89.312661,167.137518
C03797=2215.848500,71.903800,-504.076700,-102.863113,89.312661,167.137518
C03798=2216.306100,70.646200,-504.076700,-102.863113,89.312661,167.137518
C03799=2216.035600,67.030000,-504.076700,-102.863113,89.312661,167.137518
C03800=2214.885800,62.371000,-504.076700,-102.863113,89.312661,167.137518
C03801=2215.185900,59.857300,-504.076700,-102.863113,89.312661,167.137518
C03802=2216.070800,56.076700,-504.076700,-102.863113,89.312661,167.137518
C03803=2216.064600,52.308200,-504.076700,-102.863113,89.312661,167.137518
C03804=2215.795500,50.064100,-504.076700,-102.863113,89.312661,167.137518
C03805=2215.146500,46.500600,-504.076700,-102.863113,89.312661,167.137518
C03806=2216.795100,41.921000,-504.076700,-102.863113,89.312661,167.137518
C03807=2215.524300,40.173300,-504.076700,-102.863113,89.312661,167.137518
C03808=2215.817100,35.188000,-504.076700,-102.863113,89.312661,167.137518
C03809=2215.229500,33.185900,-504.076700,-102.863113,89.312661,167.137518
C03810=2216.437200,28.285200,-504.076700,-102.863113,89.312661,167.137518
C03811=2216.181700,24.390400,-504.076700,-102.863113,89.312661,167.137518
C03812=2215.618400,22.180100,-504.076700,-102.863113,89.312661,167.137518
C03813=2216.446900,16.991700,-504.076700,-102.863113,89.312661,167.137518
C03814=2216.434700,14.762000,-504.076700,-102.863113,89.312661,167.137518
C03815=2216.972500,10.736300,-504.076700,-102.863113,89.312661,167.137518
C03816=2217.092100,5.649300,-504.076700,-102.863113,89.312661,167.137518
C03817=2217.152400,3.265700,-504.076700,-102.863113,89.312661,167.137518
C03818=2215.485300,0.360200,-504.076700,-102.863113,89.312661,167.137518
C03819=2216.775300,-3.414400,-504.076700,-102.863113,89.312661,167.137518
C03820=2217.195600,-7.736900,-504.076700,-102.863113,89.312661,167.137518
C03821=2215.824400,-9.288700,-504.076700,-102.863113,89.312661,167.137518
C03822=2216.407900,-12.909500,-504.076700,-102.863113,89.312661,167.137518
C03823=2216.660600,-16.543900,-504.076700,-102.863113,89.312661,167.137518
C03824=2216.309800,-19.814400,-504.076700,-102.863113,89.312661,167.137518
C03825=2216.709700,-23.448800,-504.076700,-102.863113,89.312661,167.137518
C03826=2216.417300,-27.380700,-504.076700,-102.863113,89.312661,167.137518
C03827=2215.882300,-31.341600,-504.076700,-102.863113,89.312661,167.137518
C03828=2217.225200,-34.442000,-504.076700,-102.863113,89.312661,167.137518
C03829=2216.629200,-36.822100,-504.076700,-102.863113,89.312661,167.137518
C03830=2216.720500,-41.334700,-504.076700,-102.863113,89.312661,167.137518
C03831=2216.336100,-42.839500,-504.076700,-102.863113,89.312661,167.137518
C03832=2216.628200,-47.625900,-504.076700,-102.863113,89.312661,167.137518
C03833=2217.502000,-51.897800,-504.076700,-102.863113,89.312661,167.137518
C03834=2217.514900,-55.262800,-504.076700,-102.863113,89.312661,167.137518
C03835=2217.373400,-57.245700,-504.076700,-102.863113,89.312661,167.137518
C03836=2217.124900,-61.170300,-504.076700,-102.863113,89.312661,167.137518
C03837=2217.369200,-63.513600,-504.076700,-102.863113,89.312661,167.137518
C03838=2215.935600,-66.669100,-504.076700,-102.863113,89.312661,167.137518
C03839=2216.654700,-69.610400,-504.076700,-102.863113,89.312661,167.137518
C03840=2216.120700,-71.091900,-504.076700,-102.863113,89.312661,167.137518
C03841=2216.082800,-74.369300,-504.076700,-102.863113,89.312661,167.137518
C03842=2216.033600,-77.594900,-504.076700,-102.863113,89.312661,167.137518
C03843=2217.049900,-82.237700,-504.076700,-102.863113,89.312661,167.137518
C03844=2216.886800,-83.300300,-504.076700,-102.863113,89.312661,167.137518
C03845=2216.815000,-87.978400,-504.076700,-102.863113,89.312661,167.137518
C03846=2216.782200,-90.819000,-504.076700,-102.863113,89.312661,167.137518
C03847=2216.895900,-93.046400,-504.076700,-102.863113,89.312661,167.137518
C03848=2216.542400,-96.523900,-504.076700,-102.863113,89.312661,167.137518
C03849=2216.322600,-99.251700,-504.076700,-102.863113,89.312661,167.137518
C03850=2216.370600,-103.491300,-504.076700,-102.863113,89.312661,167.137518
C03851=2216.269200,-107.230700,-504.076700,-102.863113,89.312661,167.137518
C03852=2216.396000,-110.856300,-504.076700,-102.863113,89.312661,167.137518
C03853=2216.474800,-112.782400,-504.076700,-102.863113,89.312661,167.137518
C03854=2216.474800,-118.540500,-504.076700,-102.863113,89.312661,167.137518
C03855=2216.578700,-122.603600,-504.076700,-102.863113,89.312661,167.137518
C03856=2216.323500,-126.711100,-504.076700,-102.863113,89.312661,167.137518
C03857=2216.385600,-129.775000,-504.076700,-102.863113,89.312661,167.137518
C03858=2216.499900,-133.616000,-504.076700,-102.863113,89.312661,167.137518
C03859=2216.397100,-137.231300,-504.076700,-102.863113,89.312661,167.137518
C03860=2216.455600,-140.257700,-504.076700,-102.863113,89.312661,167.137518
C03861=2216.372700,-142.948000,-504.076700,-102.863113,89.312661,167.137518
C03862=2216.338900,-146.328800,-504.076700,-102.863113,89.312661,167.137518
C03863=2216.147500,-151.013100,-504.076700,-102.863113,89.312661,167.137518
C03864=2216.434000,-152.615800,-504.076700,-102.863113,89.312661,167.137518
C03865=2215.845300,-154.229000,-554.076700,-102.863113,89.312661,167.137518
C03866=2216.030800,-151.542800,-554.076700,-102.863113,89.312661,167.137518
C03867=2216.092300,-148.800400,-554.076700,-102.863113,89.312661,167.137518
C03868=2216.319400,-146.475800,-554.076700,-102.863113,89.312661,167.137518
C03869=2216.286200,-144.123000,-554.076700,-102.863113,89.312661,167.137518
C03870=2216.338200,-141.818900,-554.076700,-102.863113,89.312661,167.137518
C03871=2216.544000,-137.686700,-554.076700,-102.863113,89.312661,167.137518
C03872=2216.522900,-136.323200,-554.076700,-102.863113,89.312661,167.137518
C03873=2216.686100,-133.257600,-554.076700,-102.863113,89.312661,167.137518
C03874=2216.654000,-129.337200,-554.076700,-102.863113,89.312661,167.137518
C03875=2217.077100,-126.136400,-554.076700,-102.863113,89.312661,167.137518
C03876=2216.790600,-121.051200,-554.076700,-102.863113,89.312661,167.137518
C03877=2217.218300,-118.084900,-554.076700,-102.863113,89.312661,167.137518
C03878=2217.312000,-114.002400,-554.076700,-102.863113,89.312661,167.137518
C03879=2217.433700,-109.339700,-554.076700,-102.863113,89.312661,167.137518
C03880=2217.656000,-107.396800,-554.076700,-102.863113,89.312661,167.137518
C03881=2217.433000,-100.461800,-554.076700,-102.863113,89.312661,167.137518
C03882=2217.275200,-97.341500,-554.076700,-102.863113,89.312661,167.137518
C03883=2218.068000,-93.618400,-554.076700,-102.863113,89.312661,167.137518
C03884=2218.015000,-89.671400,-554.076700,-102.863113,89.312661,167.137518
C03885=2218.055100,-86.718900,-554.076700,-102.863113,89.312661,167.137518
C03886=2217.473200,-83.686300,-554.076700,-102.863113,89.312661,167.137518
C03887=2217.714900,-79.309300,-554.076700,-102.863113,89.312661,167.137518
C03888=2218.110200,-74.034800,-554.076700,-102.863113,89.312661,167.137518
C03889=2217.445200,-71.087800,-554.076700,-102.863113,89.312661,167.137518
C03890=2217.850000,-67.828900,-554.076700,-102.863113,89.312661,167.137518
C03891=2218.196300,-64.387300,-554.076700,-102.863113,89.312661,167.137518
C03892=2218.452800,-61.222000,-554.076700,-102.863113,89.312661,167.137518
C03893=2218.217900,-57.859400,-554.076700,-102.863113,89.312661,167.137518
C03894=2218.348900,-53.955600,-554.076700,-102.863113,89.312661,167.137518
C03895=2218.354500,-52.574500,-554.076700,-102.863113,89.312661,167.137518
C03896=2217.996200,-47.890600,-554.076700,-102.863113,89.312661,167.137518
C03897=2218.278900,-46.140900,-554.076700,-102.863113,89.312661,167.137518
C03898=2218.022700,-41.270900,-554.076700,-102.863113,89.312661,167.137518
C03899=2217.839700,-39.511000,-554.076700,-102.863113,89.312661,167.137518
C03900=2218.016100,-36.235600,-554.076700,-102.863113,89.312661,167.137518
C03901=2218.024100,-33.156500,-554.076700,-102.863113,89.312661,167.137518
C03902=2218.456300,-31.307100,-554.076700,-102.863113,89.312661,167.137518
C03903=2218.656000,-27.841500,-554.076700,-102.863113,89.312661,167.137518
C03904=2218.382800,-25.379300,-554.076700,-102.863113,89.312661,167.137518
C03905=2218.600600,-21.426100,-554.076700,-102.863113,89.312661,167.137518
C03906=2218.365300,-18.523700,-554.076700,-102.863113,89.312661,167.137518
C03907=2217.674500,-14.068000,-554.076700,-102.863113,89.312661,167.137518
C03908=2217.907000,-12.750200,-554.076700,-102.863113,89.312661,167.137518
C03909=2218.043600,-9.483300,-554.076700,-102.863113,89.312661,167.137518
C03910=2217.832000,-5.914300,-554.076700,-102.863113,89.312661,167.137518
C03911=2218.253400,-2.710100,-554.076700,-102.863113,89.312661,167.137518
C03912=2217.507900,-1.242900,-554.076700,-102.863113,89.312661,167.137518
C03913=2218.132300,2.684800,-554.076700,-102.863113,89.312661,167.137518
C03914=2218.032100,5.525200,-554.076700,-102.863113,89.312661,167.137518
C03915=2217.390800,8.788900,-554.076700,-102.863113,89.312661,167.137518
C03916=2218.237100,12.179400,-554.076700,-102.863113,89.312661,167.137518
C03917=2218.175400,15.755700,-554.076700,-102.863113,89.312661,167.137518
C03918=2217.434700,17.671800,-554.076700,-102.863113,89.312661,167.137518
C03919=2218.035900,22.289300,-554.076700,-102.863113,89.312661,167.137518
C03920=2217.311300,25.094600,-554.076700,-102.863113,89.312661,167.137518
C03921=2217.785000,27.188400,-554.076700,-102.863113,89.312661,167.137518
C03922=2217.217600,31.572500,-554.076700,-102.863113,89.312661,167.137518
C03923=2217.700500,33.349100,-554.076700,-102.863113,89.312661,167.137518
C03924=2217.060500,36.976400,-554.076700,-102.863113,89.312661,167.137518
C03925=2217.278200,40.078800,-554.076700,-102.863113,89.312661,167.137518
C03926=2217.586700,42.436700,-554.076700,-102.863113,89.312661,167.137518
C03927=2217.145100,45.972900,-554.076700,-102.863113,89.312661,167.137518
C03928=2217.438000,47.866400,-554.076700,-102.863113,89.312661,167.137518
C03929=2217.315500,50.859100,-554.076700,-102.863113,89.312661,167.137518
C03930=2217.508600,52.598900,-554.076700,-102.863113,89.312661,167.137518
C03931=2217.318600,56.759900,-554.076700,-102.863113,89.312661,167.137518
C03932=2217.522500,58.199900,-554.076700,-102.863113,89.312661,167.137518
C03933=2217.419700,61.688100,-554.076700,-102.863113,89.312661,167.137518
C03934=2217.351300,65.361000,-554.076700,-102.863113,89.312661,167.137518
C03935=2216.770700,66.545800,-554.076700,-102.863113,89.312661,167.137518
C03936=2217.297000,71.167000,-554.076700,-102.863113,89.312661,167.137518
C03937=2216.307900,73.267400,-554.076700,-102.863113,89.312661,167.137518
C03938=2217.071200,75.531600,-554.076700,-102.863113,89.312661,167.137518
C03939=2216.287300,77.702600,-554.076700,-102.863113,89.312661,167.137518
C03940=2216.353900,81.604100,-554.076700,-102.863113,89.312661,167.137518
C03941=2216.688500,83.493000,-554.076700,-102.863113,89.312661,167.137518
C03942=2216.770700,86.253500,-554.076700,-102.863113,89.312661,167.137518
C03943=2216.018900,88.708600,-554.076700,-102.863113,89.312661,167.137518
C03944=2216.182500,91.907500,-554.076700,-102.863113,89.312661,167.137518
C03945=2216.234700,95.968300,-554.076700,-102.863113,89.312661,167.137518
C03946=2215.706400,100.846800,-554.076700,-102.863113,89.312661,167.137518
C03947=2215.903400,102.608000,-554.076700,-102.863113,89.312661,167.137518
C03948=2216.081700,106.970900,-554.076700,-102.863113,89.312661,167.137518
C03949=2216.003200,110.390900,-554.076700,-102.863113,89.312661,167.137518
C03950=2215.690900,114.865700,-554.076700,-102.863113,89.312661,167.137518
C03951=2215.682200,117.858000,-554.076700,-102.863113,89.312661,167.137518
C03952=2215.253500,120.976000,-554.076700,-102.863113,89.312661,167.137518
C03953=2215.649800,124.738900,-554.076700,-102.863113,89.312661,167.137518
C03954=2215.331200,126.987300,-554.076700,-102.863113,89.312661,167.137518
C03955=2215.193100,130.635300,-554.076700,-102.863113,89.312661,167.137518
C03956=2215.317600,132.526300,-554.076700,-102.863113,89.312661,167.137518
C03957=2214.927800,136.778400,-554.076700,-102.863113,89.312661,167.137518
C03958=2214.786500,138.540600,-554.076700,-102.863113,89.312661,167.137518
C03959=2214.747400,142.405400,-554.076700,-102.863113,89.312661,167.137518
C03960=2215.264000,145.581000,-554.076700,-102.863113,89.312661,167.137518
C03961=2215.136700,147.696900,-554.076700,-102.863113,89.312661,167.137518
C03962=2215.109200,152.371000,-554.076700,-102.863113,89.312661,167.137518
C03963=2215.026600,156.093700,-554.076700,-102.863113,89.312661,167.137518
C03964=2214.632100,158.307600,-554.076700,-102.863113,89.312661,167.137518
C03965=2214.802500,163.078700,-554.076700,-102.863113,89.312661,167.137518
C03966=2214.248300,166.215200,-554.076700,-102.863113,89.312661,167.137518
C03967=2214.575200,170.856200,-554.076700,-102.863113,89.312661,167.137518
C03968=2214.529900,174.567100,-554.076700,-102.863113,89.312661,167.137518
C03969=2214.323900,177.868900,-554.076700,-102.863113,89.312661,167.137518
C03970=2214.200900,182.344700,-554.076700,-102.863113,89.312661,167.137518
C03971=2214.447300,186.137000,-554.076700,-102.863113,89.312661,167.137518
C03972=2214.105400,188.660700,-554.076700,-102.863113,89.312661,167.137518
C03973=2214.165700,192.211800,-554.076700,-102.863113,89.312661,167.137518
C03974=2214.182100,195.463600,-554.076700,-102.863113,89.312661,167.137518
C03975=2214.267800,200.109700,-554.076700,-102.863113,89.312661,167.137518
C03976=2214.136100,202.667800,-554.076700,-102.863113,89.312661,167.137518
C03977=2214.192500,206.310800,-554.076700,-102.863113,89.312661,167.137518
C03978=2214.077900,212.546300,-554.076700,-102.863113,89.312661,167.137518
C03979=2213.973700,214.489100,-554.076700,-102.863113,89.312661,167.137518
C03980=2214.052400,218.320600,-554.076700,-102.863113,89.312661,167.137518
C03981=2213.992800,220.807800,-554.076700,-102.863113,89.312661,167.137518
C03982=2213.896600,222.727800,-554.076700,-102.863113,89.312661,167.137518
C03983=2214.052400,226.815400,-554.076700,-102.863113,89.312661,167.137518
C03984=2214.043000,227.556900,-554.076700,-102.863113,89.312661,167.137518
C03985=2214.062200,233.401700,-554.076700,-102.863113,89.312661,167.137518
C03986=2213.854800,236.819700,-604.076700,-102.863113,89.312661,167.137518
C03987=2214.147700,232.636300,-604.076700,-102.863113,89.312661,167.137518
C03988=2214.180200,230.699500,-604.076700,-102.863113,89.312661,167.137518
C03989=2214.225300,226.783300,-604.076700,-102.863113,89.312661,167.137518
C03990=2214.196500,222.555000,-604.076700,-102.863113,89.312661,167.137518
C03991=2214.209300,219.371900,-604.076700,-102.863113,89.312661,167.137518
C03992=2214.223600,217.927300,-604.076700,-102.863113,89.312661,167.137518
C03993=2214.305800,212.992200,-604.076700,-102.863113,89.312661,167.137518
C03994=2214.235800,211.595100,-604.076700,-102.863113,89.312661,167.137518
C03995=2214.413200,205.960500,-604.076700,-102.863113,89.312661,167.137518
C03996=2214.402400,203.521200,-604.076700,-102.863113,89.312661,167.137518
C03997=2214.357700,199.539400,-604.076700,-102.863113,89.312661,167.137518
C03998=2214.617800,193.934500,-604.076700,-102.863113,89.312661,167.137518
C03999=2214.676300,190.637500,-604.076700,-102.863113,89.312661,167.137518
C04000=2214.605900,186.203900,-604.076700,-102.863113,89.312661,167.137518
C04001=2214.681900,183.258200,-604.076700,-102.863113,89.312661,167.137518
C04002=2214.906400,180.837600,-604.076700,-102.863113,89.312661,167.137518
C04003=2214.779800,177.020200,-604.076700,-102.863113,89.312661,167.137518
C04004=2214.961400,173.323200,-604.076700,-102.863113,89.312661,167.137518
C04005=2215.079900,166.661900,-604.076700,-102.863113,89.312661,167.137518
C04006=2215.427800,163.186500,-604.076700,-102.863113,89.312661,167.137518
C04007=2215.439300,158.781300,-604.076700,-102.863113,89.312661,167.137518
C04008=2215.405500,155.854500,-604.076700,-102.863113,89.312661,167.137518
C04009=2215.473800,152.247300,-604.076700,-102.863113,89.312661,167.137518
C04010=2215.553600,147.883700,-604.076700,-102.863113,89.312661,167.137518
C04011=2215.467200,143.270800,-604.076700,-102.863113,89.312661,167.137518
C04012=2215.850200,138.620000,-604.076700,-102.863113,89.312661,167.137518
C04013=2215.815700,136.272300,-604.076700,-102.863113,89.312661,167.137518
C04014=2215.828800,131.800200,-604.076700,-102.863113,89.312661,167.137518
C04015=2215.987900,127.850500,-604.076700,-102.863113,89.312661,167.137518
C04016=2215.903900,123.734800,-604.076700,-102.863113,89.312661,167.137518
C04017=2216.296000,122.317900,-604.076700,-102.863113,89.312661,167.137518
C04018=2216.159400,118.578600,-604.076700,-102.863113,89.312661,167.137518
C04019=2216.285600,115.338000,-604.076700,-102.863113,89.312661,167.137518
C04020=2216.372700,110.288600,-604.076700,-102.863113,89.312661,167.137518
C04021=2216.509000,107.801000,-604.076700,-102.863113,89.312661,167.137518
C04022=2216.520100,102.938000,-604.076700,-102.863113,89.312661,167.137518
C04023=2216.773200,97.993700,-604.076700,-102.863113,89.312661,167.137518
C04024=2216.754000,95.510200,-604.076700,-102.863113,89.312661,167.137518
C04025=2216.792000,92.305700,-604.076700,-102.863113,89.312661,167.137518
C04026=2216.990000,90.363400,-604.076700,-102.863113,89.312661,167.137518
C04027=2216.951300,86.188300,-604.076700,-102.863113,89.312661,167.137518
C04028=2217.112000,83.529500,-604.076700,-102.863113,89.312661,167.137518
C04029=2217.184100,81.108100,-604.076700,-102.863113,89.312661,167.137518
C04030=2217.220400,77.823900,-604.076700,-102.863113,89.312661,167.137518
C04031=2217.112700,74.784600,-604.076700,-102.863113,89.312661,167.137518
C04032=2217.423200,70.536700,-604.076700,-102.863113,89.312661,167.137518
C04033=2217.514200,67.590700,-604.076700,-102.863113,89.312661,167.137518
C04034=2217.308900,64.882800,-604.076700,-102.863113,89.312661,167.137518
C04035=2217.516300,62.106300,-604.076700,-102.863113,89.312661,167.137518
C04036=2217.525700,58.737100,-604.076700,-102.863113,89.312661,167.137518
C04037=2217.611400,56.232700,-604.076700,-102.863113,89.312661,167.137518
C04038=2217.651700,51.489600,-604.076700,-102.863113,89.312661,167.137518
C04039=2217.775600,49.899500,-604.076700,-102.863113,89.312661,167.137518
C04040=2217.858900,46.866700,-604.076700,-102.863113,89.312661,167.137518
C04041=2217.891300,43.600700,-604.076700,-102.863113,89.312661,167.137518
C04042=2218.053900,40.899300,-604.076700,-102.863113,89.312661,167.137518
C04043=2217.958000,36.701500,-604.076700,-102.863113,89.312661,167.137518
C04044=2218.162100,33.675700,-604.076700,-102.863113,89.312661,167.137518
C04045=2218.109800,31.032900,-604.076700,-102.863113,89.312661,167.137518
C04046=2218.166700,27.548400,-604.076700,-102.863113,89.312661,167.137518
C04047=2218.312700,24.210600,-604.076700,-102.863113,89.312661,167.137518
